LIN {X 0,Y 291.346,Z 384.19,A -85,B 0,C 180,E1 -16773.698,E2 -16773.698} C_VEL
LIN {X 0,Y 291.377,Z 384.189,A -85,B 0,C 180,E1 -16777.254,E2 -16777.254} C_VEL
LIN {X 0,Y 291.334,Z 384.196,A -85,B 0,C 180,E1 -16780.643,E2 -16780.643} C_VEL
LIN {X 0,Y 291.314,Z 384.196,A -85,B 0,C 180,E1 -16784.397,E2 -16784.397} C_VEL
LIN {X 0,Y 291.328,Z 384.196,A -85,B 0,C 180,E1 -16788.404,E2 -16788.404} C_VEL
LIN {X 0,Y 291.365,Z 384.189,A -85,B 0,C 180,E1 -16791.161,E2 -16791.161} C_VEL
LIN {X 0,Y 291.386,Z 384.191,A -85,B 0,C 180,E1 -16794.63,E2 -16794.63} C_VEL
LIN {X 0,Y 291.371,Z 384.188,A -85,B 0,C 180,E1 -16797.951,E2 -16797.951} C_VEL
LIN {X 0,Y 291.378,Z 384.187,A -85,B 0,C 180,E1 -16801.158,E2 -16801.158} C_VEL
LIN {X 0,Y 291.416,Z 384.186,A -85,B 0,C 180,E1 -16804.272,E2 -16804.272} C_VEL
LIN {X 0,Y 291.392,Z 384.185,A -85,B 0,C 180,E1 -16807.301,E2 -16807.301} C_VEL
LIN {X 0,Y 291.465,Z 384.18,A -85,B 0,C 180,E1 -16810.271,E2 -16810.271} C_VEL
LIN {X 0,Y 291.557,Z 384.166,A -85,B 0,C 180,E1 -16814.624,E2 -16814.624} C_VEL
LIN {X 0,Y 291.539,Z 384.167,A -85,B 0,C 180,E1 -16818.881,E2 -16818.881} C_VEL
LIN {X 0,Y 291.708,Z 384.147,A -85,B 0,C 180,E1 -16821.689,E2 -16821.689} C_VEL
LIN {X 0,Y 291.631,Z 384.157,A -85,B 0,C 180,E1 -16824.469,E2 -16824.469} C_VEL
LIN {X 0,Y 291.892,Z 384.124,A -85,B 0,C 180,E1 -16828.621,E2 -16828.621} C_VEL
LIN {X 0,Y 291.892,Z 384.124,A -85,B 0,C 180,E1 -16831.38,E2 -16831.38} C_VEL
LIN {X 0,Y 291.738,Z 384.142,A -85,B 0,C 180,E1 -16836.918,E2 -16836.918} C_VEL
LIN {X 0,Y 291.578,Z 384.166,A -85,B 0,C 180,E1 -16839.714,E2 -16839.714} C_VEL
LIN {X 0,Y 291.525,Z 384.172,A -85,B 0,C 180,E1 -16843.95,E2 -16843.95} C_VEL
LIN {X 0,Y 291.49,Z 384.173,A -85,B 0,C 180,E1 -16846.818,E2 -16846.818} C_VEL
LIN {X 0,Y 291.453,Z 384.18,A -85,B 0,C 180,E1 -16849.875,E2 -16849.875} C_VEL
LIN {X 0,Y 291.403,Z 384.185,A -85,B 0,C 180,E1 -16854.205,E2 -16854.205} C_VEL
LIN {X 0,Y 291.422,Z 384.184,A -85,B 0,C 180,E1 -16857.272,E2 -16857.272} C_VEL
LIN {X 0,Y 291.337,Z 384.191,A -85,B 0,C 180,E1 -16860.437,E2 -16860.437} C_VEL
LIN {X 0,Y 291.347,Z 384.194,A -85,B 0,C 180,E1 -16863.698,E2 -16863.698} C_VEL
LIN {X 0,Y 291.397,Z 384.188,A -85,B 0,C 180,E1 -16867.259,E2 -16867.259} C_VEL
LIN {X 0,Y 291.337,Z 384.192,A -85,B 0,C 180,E1 -16870.642,E2 -16870.642} C_VEL
LIN {X 0,Y 291.316,Z 384.195,A -85,B 0,C 180,E1 -16874.397,E2 -16874.397} C_VEL
LIN {X 0,Y 291.329,Z 384.193,A -85,B 0,C 180,E1 -16878.404,E2 -16878.404} C_VEL
LIN {X 0,Y 291.356,Z 384.195,A -85,B 0,C 180,E1 -16881.159,E2 -16881.159} C_VEL
LIN {X 0,Y 291.391,Z 384.186,A -85,B 0,C 180,E1 -16884.63,E2 -16884.63} C_VEL
LIN {X 0,Y 291.604,Z 384.368,A -85,B 0,C 180,E1 -16888.182,E2 -16888.182} C_VEL
LIN {X 0,Y 291.699,Z 387.226,A -85,B 0,C 180,E1 -16890.154,E2 -16890.154} C_VEL
LIN {X 0,Y 291.395,Z 391.699,A -85,B 0,C 180,E1 -16893.175,E2 -16893.175} C_VEL
LIN {X 0,Y 290.919,Z 397.87,A -85,B 0,C 180,E1 -16897.261,E2 -16897.261} C_VEL
LIN {X 0,Y 290.667,Z 402.939,A -85,B 0,C 180,E1 -16900.559,E2 -16900.559} C_VEL
LIN {X 0,Y 290.371,Z 409.272,A -85,B 0,C 180,E1 -16904.559,E2 -16904.559} C_VEL
LIN {X 0,Y 290.223,Z 413.716,A -85,B 0,C 180,E1 -16907.323,E2 -16907.323} C_VEL
LIN {X 0,Y 291.327,Z 425.543,A -85,B 0,C 180,E1 -16908.255,E2 -16908.255} C_VEL
LIN {X 0,Y 292.053,Z 433.72,A -85,B 0,C 180,E1 -16909.076,E2 -16909.076} C_VEL
LIN {X 0,Y 291.458,Z 444.808,A -85,B 0,C 180,E1 -16910.457,E2 -16910.457} C_VEL
LIN {X 0,Y 291.102,Z 453.483,A -85,B 0,C 180,E1 -16911.833,E2 -16911.833} C_VEL
LIN {X 0,Y 290.825,Z 461.477,A -85,B 0,C 180,E1 -16913.409,E2 -16913.409} C_VEL
LIN {X 0,Y 290.486,Z 468.482,A -85,B 0,C 180,E1 -16915.142,E2 -16915.142} C_VEL
LIN {X 0,Y 290.116,Z 474.952,A -85,B 0,C 180,E1 -16917.223,E2 -16917.223} C_VEL
LIN {X 0,Y 290.15,Z 479.618,A -85,B 0,C 180,E1 -16919.306,E2 -16919.306} C_VEL
LIN {X 0,Y 290.377,Z 482.726,A -85,B 0,C 180,E1 -16921.387,E2 -16921.387} C_VEL
LIN {X 0,Y 290.679,Z 483.998,A -85,B 0,C 180,E1 -16922.772,E2 -16922.772} C_VEL
LIN {X 0,Y 291.108,Z 484.656,A -85,B 0,C 180,E1 -16924.153,E2 -16924.153} C_VEL
LIN {X 0,Y 291.763,Z 484.692,A -85,B 0,C 180,E1 -16925.529,E2 -16925.529} C_VEL
LIN {X 0,Y 292.675,Z 484.009,A -85,B 0,C 180,E1 -16927.041,E2 -16927.041} C_VEL
LIN {X 0,Y 292.821,Z 483.174,A -85,B 0,C 180,E1 -16928.184,E2 -16928.184} C_VEL
LIN {X 0,Y 291.551,Z 481.327,A -85,B 0,C 180,E1 -16930.084,E2 -16930.084} C_VEL
LIN {X 0,Y 290.55,Z 478.7,A -85,B 0,C 180,E1 -16931.949,E2 -16931.949} C_VEL
LIN {X 0,Y 291.092,Z 476.418,A -85,B 0,C 180,E1 -16933.013,E2 -16933.013} C_VEL
LIN {X 0,Y 293.494,Z 470.739,A -85,B 0,C 180,E1 -16934.917,E2 -16934.917} C_VEL
LIN {X 0,Y 295.888,Z 464.445,A -85,B 0,C 180,E1 -16936.561,E2 -16936.561} C_VEL
LIN {X 0,Y 297.855,Z 458.321,A -85,B 0,C 180,E1 -16937.863,E2 -16937.863} C_VEL
LIN {X 0,Y 297.606,Z 451.062,A -85,B 0,C 180,E1 -16939.604,E2 -16939.604} C_VEL
LIN {X 0,Y 296.422,Z 443.706,A -85,B 0,C 180,E1 -16941.349,E2 -16941.349} C_VEL
LIN {X 0,Y 294.426,Z 436.045,A -85,B 0,C 180,E1 -16943.209,E2 -16943.209} C_VEL
LIN {X 0,Y 291.385,Z 427.339,A -85,B 0,C 180,E1 -16945.429,E2 -16945.429} C_VEL
LIN {X 0,Y 289.92,Z 424.703,A -85,B 0,C 180,E1 -16946.243,E2 -16946.243} C_VEL
LIN {X 0,Y 289.478,Z 422.909,A -85,B 0,C 180,E1 -16946.688,E2 -16946.688} C_VEL
LIN {X 0,Y 290.452,Z 420.929,A -85,B 0,C 180,E1 -16949.414,E2 -16949.414} C_VEL
LIN {X 0,Y 291.365,Z 419.235,A -85,B 0,C 180,E1 -16952.41,E2 -16952.41} C_VEL
LIN {X 0,Y 291.783,Z 418.234,A -85,B 0,C 180,E1 -16955.315,E2 -16955.315} C_VEL
LIN {X 0,Y 292.122,Z 417.814,A -85,B 0,C 180,E1 -16958.72,E2 -16958.72} C_VEL
LIN {X 0,Y 292.49,Z 418.223,A -85,B 0,C 180,E1 -16962.283,E2 -16962.283} C_VEL
LIN {X 0,Y 292.737,Z 418.816,A -85,B 0,C 180,E1 -16964.125,E2 -16964.125} C_VEL
LIN {X 0,Y 293.309,Z 420.913,A -85,B 0,C 180,E1 -16967.97,E2 -16967.97} C_VEL
LIN {X 0,Y 293.957,Z 423.957,A -85,B 0,C 180,E1 -16971.565,E2 -16971.565} C_VEL
LIN {X 0,Y 294.859,Z 427.941,A -85,B 0,C 180,E1 -16975.107,E2 -16975.107} C_VEL
LIN {X 0,Y 295.132,Z 430.263,A -85,B 0,C 180,E1 -16976.79,E2 -16976.79} C_VEL
LIN {X 0,Y 294.265,Z 432.986,A -85,B 0,C 180,E1 -16978.302,E2 -16978.302} C_VEL
LIN {X 0,Y 293.553,Z 434.629,A -85,B 0,C 180,E1 -16979.109,E2 -16979.109} C_VEL
LIN {X 0,Y 296.477,Z 448.571,A -85,B 0,C 180,E1 -16981.164,E2 -16981.164} C_VEL
LIN {X 0,Y 297.888,Z 460.135,A -85,B 0,C 180,E1 -16982.828,E2 -16982.828} C_VEL
LIN {X 0,Y 298.071,Z 471.015,A -85,B 0,C 180,E1 -16984.379,E2 -16984.379} C_VEL
LIN {X 0,Y 297.029,Z 480.357,A -85,B 0,C 180,E1 -16985.725,E2 -16985.725} C_VEL
LIN {X 0,Y 294.81,Z 489.886,A -85,B 0,C 180,E1 -16987.208,E2 -16987.208} C_VEL
LIN {X 0,Y 291.477,Z 500.502,A -85,B 0,C 180,E1 -16989.167,E2 -16989.167} C_VEL
LIN {X 0,Y 288.869,Z 509.05,A -85,B 0,C 180,E1 -16991.194,E2 -16991.194} C_VEL
LIN {X 0,Y 286.706,Z 516.091,A -85,B 0,C 180,E1 -16993.26,E2 -16993.26} C_VEL
LIN {X 0,Y 284.91,Z 522.618,A -85,B 0,C 180,E1 -16995.719,E2 -16995.719} C_VEL
LIN {X 0,Y 283.662,Z 527.022,A -85,B 0,C 180,E1 -16997.842,E2 -16997.842} C_VEL
LIN {X 0,Y 283.002,Z 530.416,A -85,B 0,C 180,E1 -16999.989,E2 -16999.989} C_VEL
LIN {X 0,Y 282.794,Z 532.166,A -85,B 0,C 180,E1 -17001.424,E2 -17001.424} C_VEL
LIN {X 0,Y 282.768,Z 534.128,A -85,B 0,C 180,E1 -17003.812,E2 -17003.812} C_VEL
LIN {X 0,Y 282.819,Z 534.884,A -85,B 0,C 180,E1 -17005.724,E2 -17005.724} C_VEL
LIN {X 0,Y 283.069,Z 534.95,A -85,B 0,C 180,E1 -17007.153,E2 -17007.153} C_VEL
LIN {X 0,Y 283.316,Z 534.592,A -85,B 0,C 180,E1 -17008.578,E2 -17008.578} C_VEL
LIN {X 0,Y 283.354,Z 533.788,A -85,B 0,C 180,E1 -17010,E2 -17010} C_VEL
LIN {X 0,Y 283.43,Z 532.489,A -85,B 0,C 180,E1 -17011.421,E2 -17011.421} C_VEL
LIN {X 0,Y 283.406,Z 529.608,A -85,B 0,C 180,E1 -17013.554,E2 -17013.554} C_VEL
LIN {X 0,Y 283.365,Z 525.512,A -85,B 0,C 180,E1 -17015.693,E2 -17015.693} C_VEL
LIN {X 0,Y 283.366,Z 520.078,A -85,B 0,C 180,E1 -17017.839,E2 -17017.839} C_VEL
LIN {X 0,Y 283.486,Z 513.002,A -85,B 0,C 180,E1 -17019.993,E2 -17019.993} C_VEL
LIN {X 0,Y 283.859,Z 505.706,A -85,B 0,C 180,E1 -17021.786,E2 -17021.786} C_VEL
LIN {X 0,Y 284.405,Z 496.736,A -85,B 0,C 180,E1 -17023.577,E2 -17023.577} C_VEL
LIN {X 0,Y 285.267,Z 485.479,A -85,B 0,C 180,E1 -17025.357,E2 -17025.357} C_VEL
LIN {X 0,Y 286.009,Z 474.805,A -85,B 0,C 180,E1 -17026.679,E2 -17026.679} C_VEL
LIN {X 0,Y 285.534,Z 465.102,A -85,B 0,C 180,E1 -17027.641,E2 -17027.641} C_VEL
LIN {X 0,Y 284.705,Z 452.326,A -85,B 0,C 180,E1 -17028.624,E2 -17028.624} C_VEL
LIN {X 0,Y 284.322,Z 438.684,A -85,B 0,C 180,E1 -17029.352,E2 -17029.352} C_VEL
LIN {X 0,Y 286.278,Z 425.026,A -85,B 0,C 180,E1 -17034.723,E2 -17034.723} C_VEL
LIN {X 0,Y 288.392,Z 413.702,A -85,B 0,C 180,E1 -17039.169,E2 -17039.169} C_VEL
LIN {X 0,Y 289.2,Z 409.854,A -85,B 0,C 180,E1 -17040.686,E2 -17040.686} C_VEL
LIN {X 0,Y 288.584,Z 405.721,A -85,B 0,C 180,E1 -17042.396,E2 -17042.396} C_VEL
LIN {X 0,Y 286.392,Z 395.189,A -85,B 0,C 180,E1 -17046.957,E2 -17046.957} C_VEL
LIN {X 0,Y 284.562,Z 386.236,A -85,B 0,C 180,E1 -17051.05,E2 -17051.05} C_VEL
LIN {X 0,Y 284.311,Z 385.071,A -85,B 0,C 180,E1 -17051.685,E2 -17051.685} C_VEL
LIN {X 0,Y 284.266,Z 385.073,A -85,B 0,C 180,E1 -17055.805,E2 -17055.805} C_VEL
LIN {X 0,Y 284.307,Z 385.071,A -85,B 0,C 180,E1 -17060.024,E2 -17060.024} C_VEL
LIN {X 0,Y 284.351,Z 385.064,A -85,B 0,C 180,E1 -17063.617,E2 -17063.617} C_VEL
LIN {X 0,Y 284.308,Z 385.067,A -85,B 0,C 180,E1 -17067.189,E2 -17067.189} C_VEL
LIN {X 0,Y 284.356,Z 385.064,A -85,B 0,C 180,E1 -17070.376,E2 -17070.376} C_VEL
LIN {X 0,Y 284.378,Z 385.06,A -85,B 0,C 180,E1 -17073.587,E2 -17073.587} C_VEL
LIN {X 0,Y 284.367,Z 385.06,A -85,B 0,C 180,E1 -17076.707,E2 -17076.707} C_VEL
LIN {X 0,Y 284.404,Z 385.056,A -85,B 0,C 180,E1 -17081.262,E2 -17081.262} C_VEL
LIN {X 0,Y 284.493,Z 385.045,A -85,B 0,C 180,E1 -17084.459,E2 -17084.459} C_VEL
LIN {X 0,Y 284.489,Z 385.045,A -85,B 0,C 180,E1 -17088.601,E2 -17088.601} C_VEL
LIN {X 0,Y 284.66,Z 385.026,A -85,B 0,C 180,E1 -17091.481,E2 -17091.481} C_VEL
LIN {X 0,Y 284.603,Z 385.031,A -85,B 0,C 180,E1 -17094.331,E2 -17094.331} C_VEL
LIN {X 0,Y 284.859,Z 384.998,A -85,B 0,C 180,E1 -17098.586,E2 -17098.586} C_VEL
LIN {X 0,Y 284.856,Z 385.003,A -85,B 0,C 180,E1 -17101.414,E2 -17101.414} C_VEL
LIN {X 0,Y 284.699,Z 385.021,A -85,B 0,C 180,E1 -17107.09,E2 -17107.09} C_VEL
LIN {X 0,Y 284.568,Z 385.036,A -85,B 0,C 180,E1 -17109.955,E2 -17109.955} C_VEL
LIN {X 0,Y 284.483,Z 385.046,A -85,B 0,C 180,E1 -17114.303,E2 -17114.303} C_VEL
LIN {X 0,Y 284.426,Z 385.057,A -85,B 0,C 180,E1 -17117.248,E2 -17117.248} C_VEL
LIN {X 0,Y 284.379,Z 385.059,A -85,B 0,C 180,E1 -17120.242,E2 -17120.242} C_VEL
LIN {X 0,Y 284.37,Z 385.06,A -85,B 0,C 180,E1 -17123.876,E2 -17123.876} C_VEL
LIN {X 0,Y 284.398,Z 385.06,A -85,B 0,C 180,E1 -17127.174,E2 -17127.174} C_VEL
LIN {X 0,Y 284.297,Z 385.071,A -85,B 0,C 180,E1 -17131.274,E2 -17131.274} C_VEL
LIN {X 0,Y 284.341,Z 385.065,A -85,B 0,C 180,E1 -17135.348,E2 -17135.348} C_VEL
LIN {X 0,Y 284.313,Z 385.068,A -85,B 0,C 180,E1 -17138.169,E2 -17138.169} C_VEL
LIN {X 0,Y 284.27,Z 385.072,A -85,B 0,C 180,E1 -17142.125,E2 -17142.125} C_VEL
LIN {X 0,Y 284.269,Z 385.073,A -85,B 0,C 180,E1 -17146.192,E2 -17146.192} C_VEL
LIN {X 0,Y 284.308,Z 385.068,A -85,B 0,C 180,E1 -17150.024,E2 -17150.024} C_VEL
LIN {X 0,Y 284.351,Z 385.062,A -85,B 0,C 180,E1 -17153.617,E2 -17153.617} C_VEL
LIN {X 0,Y 284.308,Z 385.068,A -85,B 0,C 180,E1 -17157.19,E2 -17157.19} C_VEL
LIN {X 0,Y 284.356,Z 385.065,A -85,B 0,C 180,E1 -17160.376,E2 -17160.376} C_VEL
LIN {X 0,Y 284.377,Z 385.059,A -85,B 0,C 180,E1 -17163.587,E2 -17163.587} C_VEL
LIN {X 0,Y 284.371,Z 385.061,A -85,B 0,C 180,E1 -17166.708,E2 -17166.708} C_VEL
LIN {X 0,Y 284.408,Z 385.055,A -85,B 0,C 180,E1 -17171.262,E2 -17171.262} C_VEL
LIN {X 0,Y 284.495,Z 385.047,A -85,B 0,C 180,E1 -17174.459,E2 -17174.459} C_VEL
LIN {X 0,Y 284.491,Z 385.046,A -85,B 0,C 180,E1 -17178.602,E2 -17178.602} C_VEL
LIN {X 0,Y 284.659,Z 385.025,A -85,B 0,C 180,E1 -17181.481,E2 -17181.481} C_VEL
LIN {X 0,Y 284.601,Z 385.033,A -85,B 0,C 180,E1 -17184.332,E2 -17184.332} C_VEL
LIN {X 0,Y 284.858,Z 385,A -85,B 0,C 180,E1 -17188.587,E2 -17188.587} C_VEL
LIN {X 0,Y 284.858,Z 385,A -85,B 0,C 180,E1 -17191.414,E2 -17191.414} C_VEL
LIN {X 0,Y 284.689,Z 385.02,A -85,B 0,C 180,E1 -17197.091,E2 -17197.091} C_VEL
LIN {X 0,Y 284.522,Z 385.045,A -85,B 0,C 180,E1 -17199.957,E2 -17199.957} C_VEL
LIN {X 0,Y 284.484,Z 385.046,A -85,B 0,C 180,E1 -17204.303,E2 -17204.303} C_VEL
LIN {X 0,Y 284.428,Z 385.054,A -85,B 0,C 180,E1 -17207.248,E2 -17207.248} C_VEL
LIN {X 0,Y 284.383,Z 385.058,A -85,B 0,C 180,E1 -17210.242,E2 -17210.242} C_VEL
LIN {X 0,Y 284.372,Z 385.062,A -85,B 0,C 180,E1 -17213.876,E2 -17213.876} C_VEL
LIN {X 0,Y 284.398,Z 385.059,A -85,B 0,C 180,E1 -17217.173,E2 -17217.173} C_VEL
LIN {X 0,Y 284.296,Z 385.071,A -85,B 0,C 180,E1 -17221.275,E2 -17221.275} C_VEL
LIN {X 0,Y 284.364,Z 385.065,A -85,B 0,C 180,E1 -17225.354,E2 -17225.354} C_VEL
LIN {X 0,Y 284.326,Z 385.064,A -85,B 0,C 180,E1 -17228.167,E2 -17228.167} C_VEL
LIN {X 0,Y 284.272,Z 385.072,A -85,B 0,C 180,E1 -17232.125,E2 -17232.125} C_VEL
LIN {X 0,Y 284.271,Z 385.071,A -85,B 0,C 180,E1 -17236.192,E2 -17236.192} C_VEL
LIN {X 0,Y 284.309,Z 385.068,A -85,B 0,C 180,E1 -17240.024,E2 -17240.024} C_VEL
LIN {X 0,Y 284.345,Z 385.064,A -85,B 0,C 180,E1 -17243.616,E2 -17243.616} C_VEL
LIN {X 0,Y 284.551,Z 385.237,A -85,B 0,C 180,E1 -17248.134,E2 -17248.134} C_VEL
LIN {X 0,Y 284.632,Z 388.458,A -85,B 0,C 180,E1 -17250.407,E2 -17250.407} C_VEL
LIN {X 0,Y 284.263,Z 393.091,A -85,B 0,C 180,E1 -17253.575,E2 -17253.575} C_VEL
LIN {X 0,Y 283.836,Z 398.85,A -85,B 0,C 180,E1 -17257.431,E2 -17257.431} C_VEL
LIN {X 0,Y 283.535,Z 404.576,A -85,B 0,C 180,E1 -17261.202,E2 -17261.202} C_VEL
LIN {X 0,Y 283.229,Z 411.459,A -85,B 0,C 180,E1 -17265.633,E2 -17265.633} C_VEL
LIN {X 0,Y 283.144,Z 414.142,A -85,B 0,C 180,E1 -17267.274,E2 -17267.274} C_VEL
LIN {X 0,Y 284.263,Z 426.11,A -85,B 0,C 180,E1 -17268.231,E2 -17268.231} C_VEL
LIN {X 0,Y 284.981,Z 433.465,A -85,B 0,C 180,E1 -17268.981,E2 -17268.981} C_VEL
LIN {X 0,Y 284.481,Z 443.471,A -85,B 0,C 180,E1 -17270.221,E2 -17270.221} C_VEL
LIN {X 0,Y 284.044,Z 453.067,A -85,B 0,C 180,E1 -17271.724,E2 -17271.724} C_VEL
LIN {X 0,Y 283.74,Z 460.853,A -85,B 0,C 180,E1 -17273.243,E2 -17273.243} C_VEL
LIN {X 0,Y 283.422,Z 468.151,A -85,B 0,C 180,E1 -17275.021,E2 -17275.021} C_VEL
LIN {X 0,Y 283.079,Z 473.868,A -85,B 0,C 180,E1 -17276.798,E2 -17276.798} C_VEL
LIN {X 0,Y 283.01,Z 478.297,A -85,B 0,C 180,E1 -17278.577,E2 -17278.577} C_VEL
LIN {X 0,Y 283.2,Z 482.167,A -85,B 0,C 180,E1 -17280.711,E2 -17280.711} C_VEL
LIN {X 0,Y 283.618,Z 484.578,A -85,B 0,C 180,E1 -17282.841,E2 -17282.841} C_VEL
LIN {X 0,Y 284.09,Z 485.407,A -85,B 0,C 180,E1 -17284.256,E2 -17284.256} C_VEL
LIN {X 0,Y 284.756,Z 485.606,A -85,B 0,C 180,E1 -17285.666,E2 -17285.666} C_VEL
LIN {X 0,Y 285.739,Z 485.062,A -85,B 0,C 180,E1 -17287.255,E2 -17287.255} C_VEL
LIN {X 0,Y 286.62,Z 484.196,A -85,B 0,C 180,E1 -17288.46,E2 -17288.46} C_VEL
LIN {X 0,Y 288.505,Z 481.559,A -85,B 0,C 180,E1 -17290.527,E2 -17290.527} C_VEL
LIN {X 0,Y 290.577,Z 477.527,A -85,B 0,C 180,E1 -17292.573,E2 -17292.573} C_VEL
LIN {X 0,Y 291.092,Z 476.418,A -85,B 0,C 180,E1 -17293.013,E2 -17293.013} C_VEL
LIN {X 0,Y 291.836,Z 473.847,A -85,B 0,C 180,E1 -17294.043,E2 -17294.043} C_VEL
LIN {X 0,Y 291.733,Z 469.418,A -85,B 0,C 180,E1 -17295.769,E2 -17295.769} C_VEL
LIN {X 0,Y 291.411,Z 463.289,A -85,B 0,C 180,E1 -17297.763,E2 -17297.763} C_VEL
LIN {X 0,Y 291.7,Z 460.914,A -85,B 0,C 180,E1 -17298.38,E2 -17298.38} C_VEL
LIN {X 0,Y 291.886,Z 455.82,A -85,B 0,C 180,E1 -17299.7,E2 -17299.7} C_VEL
LIN {X 0,Y 290.962,Z 447.353,A -85,B 0,C 180,E1 -17301.873,E2 -17301.873} C_VEL
LIN {X 0,Y 289.143,Z 439.574,A -85,B 0,C 180,E1 -17303.919,E2 -17303.919} C_VEL
LIN {X 0,Y 286.986,Z 432.608,A -85,B 0,C 180,E1 -17305.847,E2 -17305.847} C_VEL
LIN {X 0,Y 284.956,Z 427.727,A -85,B 0,C 180,E1 -17307.391,E2 -17307.391} C_VEL
LIN {X 0,Y 283.978,Z 425.851,A -85,B 0,C 180,E1 -17308.049,E2 -17308.049} C_VEL
LIN {X 0,Y 283.409,Z 423.808,A -85,B 0,C 180,E1 -17308.615,E2 -17308.615} C_VEL
LIN {X 0,Y 284.296,Z 422.222,A -85,B 0,C 180,E1 -17311.274,E2 -17311.274} C_VEL
LIN {X 0,Y 284.754,Z 421.435,A -85,B 0,C 180,E1 -17312.948,E2 -17312.948} C_VEL
LIN {X 0,Y 285.231,Z 420.555,A -85,B 0,C 180,E1 -17316.253,E2 -17316.253} C_VEL
LIN {X 0,Y 285.619,Z 420.397,A -85,B 0,C 180,E1 -17319.774,E2 -17319.774} C_VEL
LIN {X 0,Y 286.041,Z 421.202,A -85,B 0,C 180,E1 -17323.469,E2 -17323.469} C_VEL
LIN {X 0,Y 286.58,Z 423.127,A -85,B 0,C 180,E1 -17327.368,E2 -17327.368} C_VEL
LIN {X 0,Y 287.095,Z 425.487,A -85,B 0,C 180,E1 -17330.47,E2 -17330.47} C_VEL
LIN {X 0,Y 287.965,Z 429.258,A -85,B 0,C 180,E1 -17334.144,E2 -17334.144} C_VEL
LIN {X 0,Y 288.365,Z 432.715,A -85,B 0,C 180,E1 -17336.777,E2 -17336.777} C_VEL
LIN {X 0,Y 288.004,Z 434.072,A -85,B 0,C 180,E1 -17337.53,E2 -17337.53} C_VEL
LIN {X 0,Y 290.818,Z 447.57,A -85,B 0,C 180,E1 -17339.771,E2 -17339.771} C_VEL
LIN {X 0,Y 292.302,Z 461.035,A -85,B 0,C 180,E1 -17341.869,E2 -17341.869} C_VEL
LIN {X 0,Y 292.319,Z 470.96,A -85,B 0,C 180,E1 -17343.388,E2 -17343.388} C_VEL
LIN {X 0,Y 291.244,Z 480.275,A -85,B 0,C 180,E1 -17344.829,E2 -17344.829} C_VEL
LIN {X 0,Y 289.005,Z 489.552,A -85,B 0,C 180,E1 -17346.344,E2 -17346.344} C_VEL
LIN {X 0,Y 286.069,Z 498.391,A -85,B 0,C 180,E1 -17347.997,E2 -17347.997} C_VEL
LIN {X 0,Y 283.584,Z 505.824,A -85,B 0,C 180,E1 -17349.698,E2 -17349.698} C_VEL
LIN {X 0,Y 280.909,Z 513.434,A -85,B 0,C 180,E1 -17351.851,E2 -17351.851} C_VEL
LIN {X 0,Y 278.979,Z 519.262,A -85,B 0,C 180,E1 -17353.912,E2 -17353.912} C_VEL
LIN {X 0,Y 277.52,Z 524.166,A -85,B 0,C 180,E1 -17356.079,E2 -17356.079} C_VEL
LIN {X 0,Y 276.348,Z 528.017,A -85,B 0,C 180,E1 -17358.261,E2 -17358.261} C_VEL
LIN {X 0,Y 275.948,Z 530.063,A -85,B 0,C 180,E1 -17359.73,E2 -17359.73} C_VEL
LIN {X 0,Y 275.681,Z 532.878,A -85,B 0,C 180,E1 -17362.676,E2 -17362.676} C_VEL
LIN {X 0,Y 275.707,Z 533.703,A -85,B 0,C 180,E1 -17364.147,E2 -17364.147} C_VEL
LIN {X 0,Y 276.004,Z 534.05,A -85,B 0,C 180,E1 -17367.081,E2 -17367.081} C_VEL
LIN {X 0,Y 276.27,Z 533.623,A -85,B 0,C 180,E1 -17368.542,E2 -17368.542} C_VEL
LIN {X 0,Y 276.338,Z 532.687,A -85,B 0,C 180,E1 -17370,E2 -17370} C_VEL
LIN {X 0,Y 276.415,Z 531.297,A -85,B 0,C 180,E1 -17371.457,E2 -17371.457} C_VEL
LIN {X 0,Y 276.406,Z 528.256,A -85,B 0,C 180,E1 -17373.644,E2 -17373.644} C_VEL
LIN {X 0,Y 276.363,Z 523.98,A -85,B 0,C 180,E1 -17375.838,E2 -17375.838} C_VEL
LIN {X 0,Y 276.344,Z 518.268,A -85,B 0,C 180,E1 -17378.04,E2 -17378.04} C_VEL
LIN {X 0,Y 276.513,Z 510.973,A -85,B 0,C 180,E1 -17380.248,E2 -17380.248} C_VEL
LIN {X 0,Y 276.88,Z 503.352,A -85,B 0,C 180,E1 -17382.087,E2 -17382.087} C_VEL
LIN {X 0,Y 277.417,Z 494.985,A -85,B 0,C 180,E1 -17383.739,E2 -17383.739} C_VEL
LIN {X 0,Y 278.218,Z 484.775,A -85,B 0,C 180,E1 -17385.381,E2 -17385.381} C_VEL
LIN {X 0,Y 278.942,Z 473.704,A -85,B 0,C 180,E1 -17386.78,E2 -17386.78} C_VEL
LIN {X 0,Y 278.239,Z 462.1,A -85,B 0,C 180,E1 -17387.929,E2 -17387.929} C_VEL
LIN {X 0,Y 277.496,Z 449.034,A -85,B 0,C 180,E1 -17388.887,E2 -17388.887} C_VEL
LIN {X 0,Y 277.262,Z 438.473,A -85,B 0,C 180,E1 -17389.448,E2 -17389.448} C_VEL
LIN {X 0,Y 279.313,Z 424.599,A -85,B 0,C 180,E1 -17395.065,E2 -17395.065} C_VEL
LIN {X 0,Y 281.704,Z 412.566,A -85,B 0,C 180,E1 -17399.931,E2 -17399.931} C_VEL
LIN {X 0,Y 282.109,Z 409.634,A -85,B 0,C 180,E1 -17401.126,E2 -17401.126} C_VEL
LIN {X 0,Y 280.171,Z 400.291,A -85,B 0,C 180,E1 -17405.236,E2 -17405.236} C_VEL
LIN {X 0,Y 278.436,Z 391.787,A -85,B 0,C 180,E1 -17409.125,E2 -17409.125} C_VEL
LIN {X 0,Y 277.278,Z 385.948,A -85,B 0,C 180,E1 -17411.974,E2 -17411.974} C_VEL
LIN {X 0,Y 277.22,Z 385.949,A -85,B 0,C 180,E1 -17415.222,E2 -17415.222} C_VEL
LIN {X 0,Y 277.223,Z 385.95,A -85,B 0,C 180,E1 -17419.512,E2 -17419.512} C_VEL
LIN {X 0,Y 277.282,Z 385.945,A -85,B 0,C 180,E1 -17422.533,E2 -17422.533} C_VEL
LIN {X 0,Y 277.254,Z 385.95,A -85,B 0,C 180,E1 -17426.105,E2 -17426.105} C_VEL
LIN {X 0,Y 277.262,Z 385.947,A -85,B 0,C 180,E1 -17429.538,E2 -17429.538} C_VEL
LIN {X 0,Y 277.358,Z 385.933,A -85,B 0,C 180,E1 -17432.864,E2 -17432.864} C_VEL
LIN {X 0,Y 277.329,Z 385.94,A -85,B 0,C 180,E1 -17436.08,E2 -17436.08} C_VEL
LIN {X 0,Y 277.346,Z 385.935,A -85,B 0,C 180,E1 -17440.766,E2 -17440.766} C_VEL
LIN {X 0,Y 277.435,Z 385.925,A -85,B 0,C 180,E1 -17445.326,E2 -17445.326} C_VEL
LIN {X 0,Y 277.507,Z 385.918,A -85,B 0,C 180,E1 -17449.789,E2 -17449.789} C_VEL
LIN {X 0,Y 277.654,Z 385.896,A -85,B 0,C 180,E1 -17452.729,E2 -17452.729} C_VEL
LIN {X 0,Y 277.825,Z 385.875,A -85,B 0,C 180,E1 -17458.55,E2 -17458.55} C_VEL
LIN {X 0,Y 277.822,Z 385.879,A -85,B 0,C 180,E1 -17461.45,E2 -17461.45} C_VEL
LIN {X 0,Y 277.654,Z 385.9,A -85,B 0,C 180,E1 -17467.271,E2 -17467.271} C_VEL
LIN {X 0,Y 277.508,Z 385.914,A -85,B 0,C 180,E1 -17470.211,E2 -17470.211} C_VEL
LIN {X 0,Y 277.436,Z 385.924,A -85,B 0,C 180,E1 -17474.674,E2 -17474.674} C_VEL
LIN {X 0,Y 277.346,Z 385.939,A -85,B 0,C 180,E1 -17479.234,E2 -17479.234} C_VEL
LIN {X 0,Y 277.32,Z 385.938,A -85,B 0,C 180,E1 -17484.171,E2 -17484.171} C_VEL
LIN {X 0,Y 277.326,Z 385.939,A -85,B 0,C 180,E1 -17487.505,E2 -17487.505} C_VEL
LIN {X 0,Y 277.272,Z 385.945,A -85,B 0,C 180,E1 -17490.482,E2 -17490.482} C_VEL
LIN {X 0,Y 277.247,Z 385.946,A -85,B 0,C 180,E1 -17493.896,E2 -17493.896} C_VEL
LIN {X 0,Y 277.268,Z 385.945,A -85,B 0,C 180,E1 -17497.469,E2 -17497.469} C_VEL
LIN {X 0,Y 277.21,Z 385.953,A -85,B 0,C 180,E1 -17501.237,E2 -17501.237} C_VEL
LIN {X 0,Y 277.217,Z 385.952,A -85,B 0,C 180,E1 -17505.223,E2 -17505.223} C_VEL
LIN {X 0,Y 277.223,Z 385.95,A -85,B 0,C 180,E1 -17509.512,E2 -17509.512} C_VEL
LIN {X 0,Y 277.283,Z 385.945,A -85,B 0,C 180,E1 -17512.533,E2 -17512.533} C_VEL
LIN {X 0,Y 277.255,Z 385.948,A -85,B 0,C 180,E1 -17516.106,E2 -17516.106} C_VEL
LIN {X 0,Y 277.262,Z 385.944,A -85,B 0,C 180,E1 -17519.539,E2 -17519.539} C_VEL
LIN {X 0,Y 277.358,Z 385.935,A -85,B 0,C 180,E1 -17522.864,E2 -17522.864} C_VEL
LIN {X 0,Y 277.331,Z 385.939,A -85,B 0,C 180,E1 -17526.08,E2 -17526.08} C_VEL
LIN {X 0,Y 277.349,Z 385.936,A -85,B 0,C 180,E1 -17530.767,E2 -17530.767} C_VEL
LIN {X 0,Y 277.439,Z 385.923,A -85,B 0,C 180,E1 -17535.326,E2 -17535.326} C_VEL
LIN {X 0,Y 277.509,Z 385.916,A -85,B 0,C 180,E1 -17539.789,E2 -17539.789} C_VEL
LIN {X 0,Y 277.652,Z 385.897,A -85,B 0,C 180,E1 -17542.729,E2 -17542.729} C_VEL
LIN {X 0,Y 277.824,Z 385.876,A -85,B 0,C 180,E1 -17548.551,E2 -17548.551} C_VEL
LIN {X 0,Y 277.824,Z 385.876,A -85,B 0,C 180,E1 -17551.45,E2 -17551.45} C_VEL
LIN {X 0,Y 277.644,Z 385.898,A -85,B 0,C 180,E1 -17557.271,E2 -17557.271} C_VEL
LIN {X 0,Y 277.464,Z 385.922,A -85,B 0,C 180,E1 -17560.213,E2 -17560.213} C_VEL
LIN {X 0,Y 277.437,Z 385.923,A -85,B 0,C 180,E1 -17564.674,E2 -17564.674} C_VEL
LIN {X 0,Y 277.348,Z 385.936,A -85,B 0,C 180,E1 -17569.234,E2 -17569.234} C_VEL
LIN {X 0,Y 277.332,Z 385.939,A -85,B 0,C 180,E1 -17573.921,E2 -17573.921} C_VEL
LIN {X 0,Y 277.326,Z 385.942,A -85,B 0,C 180,E1 -17577.505,E2 -17577.505} C_VEL
LIN {X 0,Y 277.274,Z 385.943,A -85,B 0,C 180,E1 -17580.482,E2 -17580.482} C_VEL
LIN {X 0,Y 277.256,Z 385.948,A -85,B 0,C 180,E1 -17583.895,E2 -17583.895} C_VEL
LIN {X 0,Y 277.284,Z 385.945,A -85,B 0,C 180,E1 -17587.467,E2 -17587.467} C_VEL
LIN {X 0,Y 277.212,Z 385.955,A -85,B 0,C 180,E1 -17591.237,E2 -17591.237} C_VEL
LIN {X 0,Y 277.219,Z 385.955,A -85,B 0,C 180,E1 -17595.223,E2 -17595.223} C_VEL
LIN {X 0,Y 277.225,Z 385.952,A -85,B 0,C 180,E1 -17599.512,E2 -17599.512} C_VEL
LIN {X 0,Y 277.273,Z 385.945,A -85,B 0,C 180,E1 -17602.531,E2 -17602.531} C_VEL
LIN {X 0,Y 277.35,Z 385.935,A -85,B 0,C 180,E1 -17606.743,E2 -17606.743} C_VEL
LIN {X 0,Y 277.491,Z 386.108,A -85,B 0,C 180,E1 -17608.074,E2 -17608.074} C_VEL
LIN {X 0,Y 277.662,Z 388.205,A -85,B 0,C 180,E1 -17609.587,E2 -17609.587} C_VEL
LIN {X 0,Y 277.326,Z 392.869,A -85,B 0,C 180,E1 -17612.861,E2 -17612.861} C_VEL
LIN {X 0,Y 276.82,Z 398.646,A -85,B 0,C 180,E1 -17616.826,E2 -17616.826} C_VEL
LIN {X 0,Y 276.498,Z 404.429,A -85,B 0,C 180,E1 -17620.705,E2 -17620.705} C_VEL
LIN {X 0,Y 276.202,Z 410.21,A -85,B 0,C 180,E1 -17624.504,E2 -17624.504} C_VEL
LIN {X 0,Y 276.063,Z 414.35,A -85,B 0,C 180,E1 -17627.176,E2 -17627.176} C_VEL
LIN {X 0,Y 277.192,Z 426.674,A -85,B 0,C 180,E1 -17628.204,E2 -17628.204} C_VEL
LIN {X 0,Y 277.878,Z 433.193,A -85,B 0,C 180,E1 -17628.881,E2 -17628.881} C_VEL
LIN {X 0,Y 277.403,Z 443.381,A -85,B 0,C 180,E1 -17630.153,E2 -17630.153} C_VEL
LIN {X 0,Y 276.997,Z 452.264,A -85,B 0,C 180,E1 -17631.543,E2 -17631.543} C_VEL
LIN {X 0,Y 276.659,Z 460.106,A -85,B 0,C 180,E1 -17633.069,E2 -17633.069} C_VEL
LIN {X 0,Y 276.364,Z 467.661,A -85,B 0,C 180,E1 -17634.894,E2 -17634.894} C_VEL
LIN {X 0,Y 275.946,Z 474.682,A -85,B 0,C 180,E1 -17637.08,E2 -17637.08} C_VEL
LIN {X 0,Y 275.978,Z 479.889,A -85,B 0,C 180,E1 -17639.27,E2 -17639.27} C_VEL
LIN {X 0,Y 276.248,Z 483.495,A -85,B 0,C 180,E1 -17641.458,E2 -17641.458} C_VEL
LIN {X 0,Y 276.56,Z 485.092,A -85,B 0,C 180,E1 -17642.913,E2 -17642.913} C_VEL
LIN {X 0,Y 277.055,Z 486.079,A -85,B 0,C 180,E1 -17644.364,E2 -17644.364} C_VEL
LIN {X 0,Y 277.751,Z 486.463,A -85,B 0,C 180,E1 -17645.809,E2 -17645.809} C_VEL
LIN {X 0,Y 278.646,Z 486.248,A -85,B 0,C 180,E1 -17647.245,E2 -17647.245} C_VEL
LIN {X 0,Y 279.705,Z 485.441,A -85,B 0,C 180,E1 -17648.671,E2 -17648.671} C_VEL
LIN {X 0,Y 281.696,Z 483.079,A -85,B 0,C 180,E1 -17650.785,E2 -17650.785} C_VEL
LIN {X 0,Y 283.857,Z 479.349,A -85,B 0,C 180,E1 -17652.875,E2 -17652.875} C_VEL
LIN {X 0,Y 286.45,Z 474.156,A -85,B 0,C 180,E1 -17654.929,E2 -17654.929} C_VEL
LIN {X 0,Y 288.909,Z 468.504,A -85,B 0,C 180,E1 -17656.609,E2 -17656.609} C_VEL
LIN {X 0,Y 291.7,Z 460.914,A -85,B 0,C 180,E1 -17658.38,E2 -17658.38} C_VEL
LIN {X 0,Y 291.768,Z 458.619,A -85,B 0,C 180,E1 -17659.001,E2 -17659.001} C_VEL
LIN {X 0,Y 290.776,Z 455.722,A -85,B 0,C 180,E1 -17659.995,E2 -17659.995} C_VEL
LIN {X 0,Y 285.318,Z 448.239,A -85,B 0,C 180,E1 -17663.107,E2 -17663.107} C_VEL
LIN {X 0,Y 284.629,Z 446.126,A -85,B 0,C 180,E1 -17663.788,E2 -17663.788} C_VEL
LIN {X 0,Y 282.424,Z 437.433,A -85,B 0,C 180,E1 -17666.382,E2 -17666.382} C_VEL
LIN {X 0,Y 281.253,Z 433.862,A -85,B 0,C 180,E1 -17667.535,E2 -17667.535} C_VEL
LIN {X 0,Y 279.359,Z 429.098,A -85,B 0,C 180,E1 -17669.271,E2 -17669.271} C_VEL
LIN {X 0,Y 277.751,Z 425.837,A -85,B 0,C 180,E1 -17670.648,E2 -17670.648} C_VEL
LIN {X 0,Y 277.515,Z 424.772,A -85,B 0,C 180,E1 -17671.05,E2 -17671.05} C_VEL
LIN {X 0,Y 278.208,Z 423.653,A -85,B 0,C 180,E1 -17673.763,E2 -17673.763} C_VEL
LIN {X 0,Y 278.585,Z 423.1,A -85,B 0,C 180,E1 -17676.168,E2 -17676.168} C_VEL
LIN {X 0,Y 278.891,Z 422.96,A -85,B 0,C 180,E1 -17679.05,E2 -17679.05} C_VEL
LIN {X 0,Y 279.368,Z 423.592,A -85,B 0,C 180,E1 -17682.784,E2 -17682.784} C_VEL
LIN {X 0,Y 279.882,Z 425.349,A -85,B 0,C 180,E1 -17686.736,E2 -17686.736} C_VEL
LIN {X 0,Y 280.312,Z 427.122,A -85,B 0,C 180,E1 -17689.316,E2 -17689.316} C_VEL
LIN {X 0,Y 281.058,Z 430.656,A -85,B 0,C 180,E1 -17693.147,E2 -17693.147} C_VEL
LIN {X 0,Y 281.642,Z 433.418,A -85,B 0,C 180,E1 -17695.383,E2 -17695.383} C_VEL
LIN {X 0,Y 283.578,Z 438.057,A -85,B 0,C 180,E1 -17696.626,E2 -17696.626} C_VEL
LIN {X 0,Y 285.414,Z 447.46,A -85,B 0,C 180,E1 -17698.384,E2 -17698.384} C_VEL
LIN {X 0,Y 286.667,Z 459.662,A -85,B 0,C 180,E1 -17700.465,E2 -17700.465} C_VEL
LIN {X 0,Y 286.74,Z 470.393,A -85,B 0,C 180,E1 -17702.245,E2 -17702.245} C_VEL
LIN {X 0,Y 285.742,Z 479.369,A -85,B 0,C 180,E1 -17703.722,E2 -17703.722} C_VEL
LIN {X 0,Y 283.247,Z 489.377,A -85,B 0,C 180,E1 -17705.442,E2 -17705.442} C_VEL
LIN {X 0,Y 280.192,Z 498.046,A -85,B 0,C 180,E1 -17707.121,E2 -17707.121} C_VEL
LIN {X 0,Y 277.99,Z 503.959,A -85,B 0,C 180,E1 -17708.495,E2 -17708.495} C_VEL
LIN {X 0,Y 275.108,Z 511.518,A -85,B 0,C 180,E1 -17710.603,E2 -17710.603} C_VEL
LIN {X 0,Y 272.802,Z 517.677,A -85,B 0,C 180,E1 -17712.766,E2 -17712.766} C_VEL
LIN {X 0,Y 271.127,Z 522.685,A -85,B 0,C 180,E1 -17714.976,E2 -17714.976} C_VEL
LIN {X 0,Y 269.72,Z 526.65,A -85,B 0,C 180,E1 -17717.204,E2 -17717.204} C_VEL
LIN {X 0,Y 268.914,Z 529.655,A -85,B 0,C 180,E1 -17719.458,E2 -17719.458} C_VEL
LIN {X 0,Y 268.606,Z 532.276,A -85,B 0,C 180,E1 -17722.483,E2 -17722.483} C_VEL
LIN {X 0,Y 268.649,Z 532.958,A -85,B 0,C 180,E1 -17723.993,E2 -17723.993} C_VEL
LIN {X 0,Y 268.941,Z 533.136,A -85,B 0,C 180,E1 -17727.004,E2 -17727.004} C_VEL
LIN {X 0,Y 269.236,Z 532.573,A -85,B 0,C 180,E1 -17728.504,E2 -17728.504} C_VEL
LIN {X 0,Y 269.326,Z 531.549,A -85,B 0,C 180,E1 -17730,E2 -17730} C_VEL
LIN {X 0,Y 269.405,Z 529.107,A -85,B 0,C 180,E1 -17732.242,E2 -17732.242} C_VEL
LIN {X 0,Y 269.378,Z 525.487,A -85,B 0,C 180,E1 -17734.489,E2 -17734.489} C_VEL
LIN {X 0,Y 269.353,Z 520.132,A -85,B 0,C 180,E1 -17736.896,E2 -17736.896} C_VEL
LIN {X 0,Y 269.382,Z 514.048,A -85,B 0,C 180,E1 -17739.006,E2 -17739.006} C_VEL
LIN {X 0,Y 269.632,Z 507.318,A -85,B 0,C 180,E1 -17740.893,E2 -17740.893} C_VEL
LIN {X 0,Y 270.111,Z 499.06,A -85,B 0,C 180,E1 -17742.777,E2 -17742.777} C_VEL
LIN {X 0,Y 270.757,Z 488.774,A -85,B 0,C 180,E1 -17744.66,E2 -17744.66} C_VEL
LIN {X 0,Y 271.551,Z 478.517,A -85,B 0,C 180,E1 -17746.154,E2 -17746.154} C_VEL
LIN {X 0,Y 271.803,Z 472.185,A -85,B 0,C 180,E1 -17746.92,E2 -17746.92} C_VEL
LIN {X 0,Y 270.97,Z 459.849,A -85,B 0,C 180,E1 -17748.134,E2 -17748.134} C_VEL
LIN {X 0,Y 270.301,Z 447.101,A -85,B 0,C 180,E1 -17749.064,E2 -17749.064} C_VEL
LIN {X 0,Y 270.199,Z 438.12,A -85,B 0,C 180,E1 -17749.565,E2 -17749.565} C_VEL
LIN {X 0,Y 272.322,Z 424.167,A -85,B 0,C 180,E1 -17755.409,E2 -17755.409} C_VEL
LIN {X 0,Y 275.005,Z 411.437,A -85,B 0,C 180,E1 -17760.738,E2 -17760.738} C_VEL
LIN {X 0,Y 274.54,Z 407.743,A -85,B 0,C 180,E1 -17762.352,E2 -17762.352} C_VEL
LIN {X 0,Y 272.448,Z 397.845,A -85,B 0,C 180,E1 -17766.901,E2 -17766.901} C_VEL
LIN {X 0,Y 270.65,Z 389.001,A -85,B 0,C 180,E1 -17771.145,E2 -17771.145} C_VEL
LIN {X 0,Y 270.227,Z 386.827,A -85,B 0,C 180,E1 -17772.248,E2 -17772.248} C_VEL
LIN {X 0,Y 270.173,Z 386.828,A -85,B 0,C 180,E1 -17776.749,E2 -17776.749} C_VEL
LIN {X 0,Y 270.222,Z 386.823,A -85,B 0,C 180,E1 -17781.283,E2 -17781.283} C_VEL
LIN {X 0,Y 270.215,Z 386.822,A -85,B 0,C 180,E1 -17785.096,E2 -17785.096} C_VEL
LIN {X 0,Y 270.2,Z 386.825,A -85,B 0,C 180,E1 -17789.13,E2 -17789.13} C_VEL
LIN {X 0,Y 270.264,Z 386.82,A -85,B 0,C 180,E1 -17792.146,E2 -17792.146} C_VEL
LIN {X 0,Y 270.278,Z 386.816,A -85,B 0,C 180,E1 -17795.519,E2 -17795.519} C_VEL
LIN {X 0,Y 270.302,Z 386.814,A -85,B 0,C 180,E1 -17800.244,E2 -17800.244} C_VEL
LIN {X 0,Y 270.403,Z 386.799,A -85,B 0,C 180,E1 -17804.935,E2 -17804.935} C_VEL
LIN {X 0,Y 270.442,Z 386.798,A -85,B 0,C 180,E1 -17809.519,E2 -17809.519} C_VEL
LIN {X 0,Y 270.612,Z 386.773,A -85,B 0,C 180,E1 -17812.539,E2 -17812.539} C_VEL
LIN {X 0,Y 270.791,Z 386.751,A -85,B 0,C 180,E1 -17818.513,E2 -17818.513} C_VEL
LIN {X 0,Y 270.788,Z 386.755,A -85,B 0,C 180,E1 -17821.487,E2 -17821.487} C_VEL
LIN {X 0,Y 270.612,Z 386.776,A -85,B 0,C 180,E1 -17827.461,E2 -17827.461} C_VEL
LIN {X 0,Y 270.443,Z 386.794,A -85,B 0,C 180,E1 -17830.481,E2 -17830.481} C_VEL
LIN {X 0,Y 270.404,Z 386.803,A -85,B 0,C 180,E1 -17835.065,E2 -17835.065} C_VEL
LIN {X 0,Y 270.302,Z 386.813,A -85,B 0,C 180,E1 -17839.756,E2 -17839.756} C_VEL
LIN {X 0,Y 270.275,Z 386.816,A -85,B 0,C 180,E1 -17844.586,E2 -17844.586} C_VEL
LIN {X 0,Y 270.272,Z 386.816,A -85,B 0,C 180,E1 -17847.909,E2 -17847.909} C_VEL
LIN {X 0,Y 270.185,Z 386.829,A -85,B 0,C 180,E1 -17851.348,E2 -17851.348} C_VEL
LIN {X 0,Y 270.202,Z 386.828,A -85,B 0,C 180,E1 -17854.906,E2 -17854.906} C_VEL
LIN {X 0,Y 270.198,Z 386.829,A -85,B 0,C 180,E1 -17858.711,E2 -17858.711} C_VEL
LIN {X 0,Y 270.172,Z 386.829,A -85,B 0,C 180,E1 -17863.251,E2 -17863.251} C_VEL
LIN {X 0,Y 270.175,Z 386.829,A -85,B 0,C 180,E1 -17867.443,E2 -17867.443} C_VEL
LIN {X 0,Y 270.207,Z 386.823,A -85,B 0,C 180,E1 -17871.374,E2 -17871.374} C_VEL
LIN {X 0,Y 270.216,Z 386.824,A -85,B 0,C 180,E1 -17875.097,E2 -17875.097} C_VEL
LIN {X 0,Y 270.201,Z 386.824,A -85,B 0,C 180,E1 -17879.131,E2 -17879.131} C_VEL
LIN {X 0,Y 270.264,Z 386.819,A -85,B 0,C 180,E1 -17882.147,E2 -17882.147} C_VEL
LIN {X 0,Y 270.279,Z 386.815,A -85,B 0,C 180,E1 -17885.519,E2 -17885.519} C_VEL
LIN {X 0,Y 270.305,Z 386.815,A -85,B 0,C 180,E1 -17890.245,E2 -17890.245} C_VEL
LIN {X 0,Y 270.407,Z 386.799,A -85,B 0,C 180,E1 -17894.936,E2 -17894.936} C_VEL
LIN {X 0,Y 270.444,Z 386.795,A -85,B 0,C 180,E1 -17899.519,E2 -17899.519} C_VEL
LIN {X 0,Y 270.61,Z 386.776,A -85,B 0,C 180,E1 -17902.539,E2 -17902.539} C_VEL
LIN {X 0,Y 270.79,Z 386.753,A -85,B 0,C 180,E1 -17908.513,E2 -17908.513} C_VEL
LIN {X 0,Y 270.79,Z 386.753,A -85,B 0,C 180,E1 -17911.487,E2 -17911.487} C_VEL
LIN {X 0,Y 270.601,Z 386.777,A -85,B 0,C 180,E1 -17917.462,E2 -17917.462} C_VEL
LIN {X 0,Y 270.416,Z 386.798,A -85,B 0,C 180,E1 -17920.482,E2 -17920.482} C_VEL
LIN {X 0,Y 270.406,Z 386.799,A -85,B 0,C 180,E1 -17925.065,E2 -17925.065} C_VEL
LIN {X 0,Y 270.305,Z 386.815,A -85,B 0,C 180,E1 -17929.756,E2 -17929.756} C_VEL
LIN {X 0,Y 270.277,Z 386.816,A -85,B 0,C 180,E1 -17934.586,E2 -17934.586} C_VEL
LIN {X 0,Y 270.272,Z 386.817,A -85,B 0,C 180,E1 -17937.909,E2 -17937.909} C_VEL
LIN {X 0,Y 270.186,Z 386.829,A -85,B 0,C 180,E1 -17941.348,E2 -17941.348} C_VEL
LIN {X 0,Y 270.217,Z 386.824,A -85,B 0,C 180,E1 -17944.904,E2 -17944.904} C_VEL
LIN {X 0,Y 270.225,Z 386.821,A -85,B 0,C 180,E1 -17948.717,E2 -17948.717} C_VEL
LIN {X 0,Y 270.174,Z 386.833,A -85,B 0,C 180,E1 -17953.251,E2 -17953.251} C_VEL
LIN {X 0,Y 270.177,Z 386.83,A -85,B 0,C 180,E1 -17957.442,E2 -17957.442} C_VEL
LIN {X 0,Y 270.209,Z 386.827,A -85,B 0,C 180,E1 -17961.374,E2 -17961.374} C_VEL
LIN {X 0,Y 270.256,Z 386.821,A -85,B 0,C 180,E1 -17965.102,E2 -17965.102} C_VEL
LIN {X 0,Y 270.459,Z 386.966,A -85,B 0,C 180,E1 -17968.031,E2 -17968.031} C_VEL
LIN {X 0,Y 270.595,Z 389.258,A -85,B 0,C 180,E1 -17969.708,E2 -17969.708} C_VEL
LIN {X 0,Y 270.262,Z 393.794,A -85,B 0,C 180,E1 -17972.93,E2 -17972.93} C_VEL
LIN {X 0,Y 269.733,Z 399.593,A -85,B 0,C 180,E1 -17976.994,E2 -17976.994} C_VEL
LIN {X 0,Y 269.409,Z 405.406,A -85,B 0,C 180,E1 -17980.969,E2 -17980.969} C_VEL
LIN {X 0,Y 269.077,Z 411.607,A -85,B 0,C 180,E1 -17985.107,E2 -17985.107} C_VEL
LIN {X 0,Y 268.976,Z 414.665,A -85,B 0,C 180,E1 -17987.12,E2 -17987.12} C_VEL
LIN {X 0,Y 270.105,Z 427.105,A -85,B 0,C 180,E1 -17988.176,E2 -17988.176} C_VEL
LIN {X 0,Y 270.727,Z 434.397,A -85,B 0,C 180,E1 -17988.962,E2 -17988.962} C_VEL
LIN {X 0,Y 270.224,Z 444.346,A -85,B 0,C 180,E1 -17990.267,E2 -17990.267} C_VEL
LIN {X 0,Y 269.82,Z 453.707,A -85,B 0,C 180,E1 -17991.806,E2 -17991.806} C_VEL
LIN {X 0,Y 269.522,Z 462.579,A -85,B 0,C 180,E1 -17993.637,E2 -17993.637} C_VEL
LIN {X 0,Y 269.119,Z 469.773,A -85,B 0,C 180,E1 -17995.507,E2 -17995.507} C_VEL
LIN {X 0,Y 268.847,Z 475.482,A -85,B 0,C 180,E1 -17997.378,E2 -17997.378} C_VEL
LIN {X 0,Y 268.875,Z 479.886,A -85,B 0,C 180,E1 -17999.251,E2 -17999.251} C_VEL
LIN {X 0,Y 269.168,Z 483.761,A -85,B 0,C 180,E1 -18001.496,E2 -18001.496} C_VEL
LIN {X 0,Y 269.503,Z 485.552,A -85,B 0,C 180,E1 -18002.99,E2 -18002.99} C_VEL
LIN {X 0,Y 270.008,Z 486.736,A -85,B 0,C 180,E1 -18004.479,E2 -18004.479} C_VEL
LIN {X 0,Y 270.748,Z 487.291,A -85,B 0,C 180,E1 -18005.96,E2 -18005.96} C_VEL
LIN {X 0,Y 271.674,Z 487.246,A -85,B 0,C 180,E1 -18007.432,E2 -18007.432} C_VEL
LIN {X 0,Y 272.784,Z 486.627,A -85,B 0,C 180,E1 -18008.893,E2 -18008.893} C_VEL
LIN {X 0,Y 274.132,Z 485.412,A -85,B 0,C 180,E1 -18010.338,E2 -18010.338} C_VEL
LIN {X 0,Y 276.345,Z 482.499,A -85,B 0,C 180,E1 -18012.484,E2 -18012.484} C_VEL
LIN {X 0,Y 278.938,Z 478.161,A -85,B 0,C 180,E1 -18014.593,E2 -18014.593} C_VEL
LIN {X 0,Y 281.867,Z 472.266,A -85,B 0,C 180,E1 -18016.663,E2 -18016.663} C_VEL
LIN {X 0,Y 284.701,Z 465.994,A -85,B 0,C 180,E1 -18018.345,E2 -18018.345} C_VEL
LIN {X 0,Y 285.869,Z 462.744,A -85,B 0,C 180,E1 -18019.114,E2 -18019.114} C_VEL
LIN {X 0,Y 285.886,Z 455.244,A -85,B 0,C 180,E1 -18021.223,E2 -18021.223} C_VEL
LIN {X 0,Y 284.875,Z 447.377,A -85,B 0,C 180,E1 -18023.424,E2 -18023.424} C_VEL
LIN {X 0,Y 284.629,Z 446.126,A -85,B 0,C 180,E1 -18023.788,E2 -18023.788} C_VEL
LIN {X 0,Y 283.493,Z 443.29,A -85,B 0,C 180,E1 -18024.805,E2 -18024.805} C_VEL
LIN {X 0,Y 281.685,Z 441.237,A -85,B 0,C 180,E1 -18025.874,E2 -18025.874} C_VEL
LIN {X 0,Y 276.418,Z 436.644,A -85,B 0,C 180,E1 -18028.839,E2 -18028.839} C_VEL
LIN {X 0,Y 275.568,Z 435.028,A -85,B 0,C 180,E1 -18029.579,E2 -18029.579} C_VEL
LIN {X 0,Y 274.131,Z 431.115,A -85,B 0,C 180,E1 -18031.276,E2 -18031.276} C_VEL
LIN {X 0,Y 271.913,Z 426.976,A -85,B 0,C 180,E1 -18033.735,E2 -18033.735} C_VEL
LIN {X 0,Y 271.632,Z 426.02,A -85,B 0,C 180,E1 -18034.234,E2 -18034.234} C_VEL
LIN {X 0,Y 272.016,Z 425.574,A -85,B 0,C 180,E1 -18036.779,E2 -18036.779} C_VEL
LIN {X 0,Y 272.384,Z 425.673,A -85,B 0,C 180,E1 -18040.169,E2 -18040.169} C_VEL
LIN {X 0,Y 272.888,Z 426.584,A -85,B 0,C 180,E1 -18043.853,E2 -18043.853} C_VEL
LIN {X 0,Y 273.166,Z 427.624,A -85,B 0,C 180,E1 -18046.086,E2 -18046.086} C_VEL
LIN {X 0,Y 273.496,Z 428.906,A -85,B 0,C 180,E1 -18048.177,E2 -18048.177} C_VEL
LIN {X 0,Y 274.174,Z 432.113,A -85,B 0,C 180,E1 -18051.983,E2 -18051.983} C_VEL
LIN {X 0,Y 277.109,Z 437.71,A -85,B 0,C 180,E1 -18054.251,E2 -18054.251} C_VEL
LIN {X 0,Y 278.027,Z 438.934,A -85,B 0,C 180,E1 -18054.821,E2 -18054.821} C_VEL
LIN {X 0,Y 279.769,Z 443.934,A -85,B 0,C 180,E1 -18056.184,E2 -18056.184} C_VEL
LIN {X 0,Y 281.094,Z 454.982,A -85,B 0,C 180,E1 -18058.328,E2 -18058.328} C_VEL
LIN {X 0,Y 281.394,Z 466.911,A -85,B 0,C 180,E1 -18060.485,E2 -18060.485} C_VEL
LIN {X 0,Y 280.714,Z 475.901,A -85,B 0,C 180,E1 -18062.09,E2 -18062.09} C_VEL
LIN {X 0,Y 279.269,Z 483.7,A -85,B 0,C 180,E1 -18063.468,E2 -18063.468} C_VEL
LIN {X 0,Y 276.326,Z 492.929,A -85,B 0,C 180,E1 -18065.187,E2 -18065.187} C_VEL
LIN {X 0,Y 272.496,Z 502.228,A -85,B 0,C 180,E1 -18067.24,E2 -18067.24} C_VEL
LIN {X 0,Y 269.46,Z 509.856,A -85,B 0,C 180,E1 -18069.384,E2 -18069.384} C_VEL
LIN {X 0,Y 266.76,Z 516.159,A -85,B 0,C 180,E1 -18071.569,E2 -18071.569} C_VEL
LIN {X 0,Y 264.745,Z 521.255,A -85,B 0,C 180,E1 -18073.815,E2 -18073.815} C_VEL
LIN {X 0,Y 262.772,Z 526.466,A -85,B 0,C 180,E1 -18076.859,E2 -18076.859} C_VEL
LIN {X 0,Y 261.893,Z 529.266,A -85,B 0,C 180,E1 -18079.172,E2 -18079.172} C_VEL
LIN {X 0,Y 261.528,Z 531.606,A -85,B 0,C 180,E1 -18082.278,E2 -18082.278} C_VEL
LIN {X 0,Y 261.572,Z 532.203,A -85,B 0,C 180,E1 -18083.83,E2 -18083.83} C_VEL
LIN {X 0,Y 261.625,Z 532.382,A -85,B 0,C 180,E1 -18085.377,E2 -18085.377} C_VEL
LIN {X 0,Y 261.896,Z 532.138,A -85,B 0,C 180,E1 -18086.923,E2 -18086.923} C_VEL
LIN {X 0,Y 262.206,Z 531.492,A -85,B 0,C 180,E1 -18088.464,E2 -18088.464} C_VEL
LIN {X 0,Y 262.321,Z 530.37,A -85,B 0,C 180,E1 -18090,E2 -18090} C_VEL
LIN {X 0,Y 262.437,Z 527.747,A -85,B 0,C 180,E1 -18092.302,E2 -18092.302} C_VEL
LIN {X 0,Y 262.38,Z 523.899,A -85,B 0,C 180,E1 -18094.609,E2 -18094.609} C_VEL
LIN {X 0,Y 262.365,Z 518.37,A -85,B 0,C 180,E1 -18097.06,E2 -18097.06} C_VEL
LIN {X 0,Y 262.382,Z 511.957,A -85,B 0,C 180,E1 -18099.248,E2 -18099.248} C_VEL
LIN {X 0,Y 262.757,Z 503.346,A -85,B 0,C 180,E1 -18101.572,E2 -18101.572} C_VEL
LIN {X 0,Y 263.266,Z 494.311,A -85,B 0,C 180,E1 -18103.508,E2 -18103.508} C_VEL
LIN {X 0,Y 264.054,Z 484.305,A -85,B 0,C 180,E1 -18105.238,E2 -18105.238} C_VEL
LIN {X 0,Y 264.718,Z 474.643,A -85,B 0,C 180,E1 -18106.583,E2 -18106.583} C_VEL
LIN {X 0,Y 264.253,Z 465.672,A -85,B 0,C 180,E1 -18107.589,E2 -18107.589} C_VEL
LIN {X 0,Y 263.408,Z 452.012,A -85,B 0,C 180,E1 -18108.774,E2 -18108.774} C_VEL
LIN {X 0,Y 263.06,Z 439.974,A -85,B 0,C 180,E1 -18109.509,E2 -18109.509} C_VEL
LIN {X 0,Y 263.113,Z 437.942,A -85,B 0,C 180,E1 -18109.606,E2 -18109.606} C_VEL
LIN {X 0,Y 265.088,Z 425.284,A -85,B 0,C 180,E1 -18115.099,E2 -18115.099} C_VEL
LIN {X 0,Y 267.901,Z 412.188,A -85,B 0,C 180,E1 -18120.767,E2 -18120.767} C_VEL
LIN {X 0,Y 267.573,Z 409.032,A -85,B 0,C 180,E1 -18122.189,E2 -18122.189} C_VEL
LIN {X 0,Y 265.613,Z 399.923,A -85,B 0,C 180,E1 -18126.446,E2 -18126.446} C_VEL
LIN {X 0,Y 264.077,Z 392.378,A -85,B 0,C 180,E1 -18130.169,E2 -18130.169} C_VEL
LIN {X 0,Y 263.204,Z 387.702,A -85,B 0,C 180,E1 -18132.564,E2 -18132.564} C_VEL
LIN {X 0,Y 263.13,Z 387.709,A -85,B 0,C 180,E1 -18136.149,E2 -18136.149} C_VEL
LIN {X 0,Y 263.116,Z 387.712,A -85,B 0,C 180,E1 -18140.129,E2 -18140.129} C_VEL
LIN {X 0,Y 263.188,Z 387.702,A -85,B 0,C 180,E1 -18144.022,E2 -18144.022} C_VEL
LIN {X 0,Y 263.134,Z 387.707,A -85,B 0,C 180,E1 -18147.712,E2 -18147.712} C_VEL
LIN {X 0,Y 263.196,Z 387.701,A -85,B 0,C 180,E1 -18151.785,E2 -18151.785} C_VEL
LIN {X 0,Y 263.226,Z 387.693,A -85,B 0,C 180,E1 -18155.2,E2 -18155.2} C_VEL
LIN {X 0,Y 263.264,Z 387.693,A -85,B 0,C 180,E1 -18159.693,E2 -18159.693} C_VEL
LIN {X 0,Y 263.352,Z 387.678,A -85,B 0,C 180,E1 -18164.522,E2 -18164.522} C_VEL
LIN {X 0,Y 263.375,Z 387.677,A -85,B 0,C 180,E1 -18169.234,E2 -18169.234} C_VEL
LIN {X 0,Y 263.574,Z 387.65,A -85,B 0,C 180,E1 -18172.338,E2 -18172.338} C_VEL
LIN {X 0,Y 263.755,Z 387.627,A -85,B 0,C 180,E1 -18178.473,E2 -18178.473} C_VEL
LIN {X 0,Y 263.752,Z 387.632,A -85,B 0,C 180,E1 -18181.527,E2 -18181.527} C_VEL
LIN {X 0,Y 263.574,Z 387.651,A -85,B 0,C 180,E1 -18187.662,E2 -18187.662} C_VEL
LIN {X 0,Y 263.376,Z 387.676,A -85,B 0,C 180,E1 -18190.766,E2 -18190.766} C_VEL
LIN {X 0,Y 263.352,Z 387.68,A -85,B 0,C 180,E1 -18195.478,E2 -18195.478} C_VEL
LIN {X 0,Y 263.264,Z 387.689,A -85,B 0,C 180,E1 -18200.307,E2 -18200.307} C_VEL
LIN {X 0,Y 263.209,Z 387.697,A -85,B 0,C 180,E1 -18205.291,E2 -18205.291} C_VEL
LIN {X 0,Y 263.18,Z 387.702,A -85,B 0,C 180,E1 -18208.73,E2 -18208.73} C_VEL
LIN {X 0,Y 263.134,Z 387.706,A -85,B 0,C 180,E1 -18212.288,E2 -18212.288} C_VEL
LIN {X 0,Y 263.183,Z 387.702,A -85,B 0,C 180,E1 -18216.764,E2 -18216.764} C_VEL
LIN {X 0,Y 263.125,Z 387.705,A -85,B 0,C 180,E1 -18221.594,E2 -18221.594} C_VEL
LIN {X 0,Y 263.128,Z 387.706,A -85,B 0,C 180,E1 -18226.017,E2 -18226.017} C_VEL
LIN {X 0,Y 263.116,Z 387.708,A -85,B 0,C 180,E1 -18230.13,E2 -18230.13} C_VEL
LIN {X 0,Y 263.189,Z 387.699,A -85,B 0,C 180,E1 -18234.022,E2 -18234.022} C_VEL
LIN {X 0,Y 263.134,Z 387.705,A -85,B 0,C 180,E1 -18237.712,E2 -18237.712} C_VEL
LIN {X 0,Y 263.199,Z 387.697,A -85,B 0,C 180,E1 -18241.785,E2 -18241.785} C_VEL
LIN {X 0,Y 263.227,Z 387.694,A -85,B 0,C 180,E1 -18245.201,E2 -18245.201} C_VEL
LIN {X 0,Y 263.271,Z 387.688,A -85,B 0,C 180,E1 -18249.694,E2 -18249.694} C_VEL
LIN {X 0,Y 263.354,Z 387.68,A -85,B 0,C 180,E1 -18254.522,E2 -18254.522} C_VEL
LIN {X 0,Y 263.376,Z 387.675,A -85,B 0,C 180,E1 -18259.235,E2 -18259.235} C_VEL
LIN {X 0,Y 263.572,Z 387.654,A -85,B 0,C 180,E1 -18262.339,E2 -18262.339} C_VEL
LIN {X 0,Y 263.754,Z 387.63,A -85,B 0,C 180,E1 -18268.473,E2 -18268.473} C_VEL
LIN {X 0,Y 263.754,Z 387.63,A -85,B 0,C 180,E1 -18271.527,E2 -18271.527} C_VEL
LIN {X 0,Y 263.561,Z 387.655,A -85,B 0,C 180,E1 -18277.662,E2 -18277.662} C_VEL
LIN {X 0,Y 263.358,Z 387.677,A -85,B 0,C 180,E1 -18280.767,E2 -18280.767} C_VEL
LIN {X 0,Y 263.354,Z 387.68,A -85,B 0,C 180,E1 -18285.478,E2 -18285.478} C_VEL
LIN {X 0,Y 263.267,Z 387.688,A -85,B 0,C 180,E1 -18290.307,E2 -18290.307} C_VEL
LIN {X 0,Y 263.211,Z 387.698,A -85,B 0,C 180,E1 -18295.291,E2 -18295.291} C_VEL
LIN {X 0,Y 263.178,Z 387.699,A -85,B 0,C 180,E1 -18298.73,E2 -18298.73} C_VEL
LIN {X 0,Y 263.136,Z 387.705,A -85,B 0,C 180,E1 -18302.288,E2 -18302.288} C_VEL
LIN {X 0,Y 263.19,Z 387.699,A -85,B 0,C 180,E1 -18305.978,E2 -18305.978} C_VEL
LIN {X 0,Y 263.118,Z 387.708,A -85,B 0,C 180,E1 -18309.871,E2 -18309.871} C_VEL
LIN {X 0,Y 263.13,Z 387.706,A -85,B 0,C 180,E1 -18313.983,E2 -18313.983} C_VEL
LIN {X 0,Y 263.127,Z 387.705,A -85,B 0,C 180,E1 -18318.406,E2 -18318.406} C_VEL
LIN {X 0,Y 263.192,Z 387.701,A -85,B 0,C 180,E1 -18323.235,E2 -18323.235} C_VEL
LIN {X 0,Y 263.43,Z 387.862,A -85,B 0,C 180,E1 -18328.01,E2 -18328.01} C_VEL
LIN {X 0,Y 263.504,Z 391.114,A -85,B 0,C 180,E1 -18330.434,E2 -18330.434} C_VEL
LIN {X 0,Y 262.944,Z 397.015,A -85,B 0,C 180,E1 -18334.681,E2 -18334.681} C_VEL
LIN {X 0,Y 262.466,Z 404.048,A -85,B 0,C 180,E1 -18339.629,E2 -18339.629} C_VEL
LIN {X 0,Y 262.048,Z 411.101,A -85,B 0,C 180,E1 -18344.443,E2 -18344.443} C_VEL
LIN {X 0,Y 261.89,Z 415.005,A -85,B 0,C 180,E1 -18347.061,E2 -18347.061} C_VEL
LIN {X 0,Y 263.103,Z 428.221,A -85,B 0,C 180,E1 -18348.248,E2 -18348.248} C_VEL
LIN {X 0,Y 263.645,Z 433.761,A -85,B 0,C 180,E1 -18348.857,E2 -18348.857} C_VEL
LIN {X 0,Y 263.148,Z 443.972,A -85,B 0,C 180,E1 -18350.197,E2 -18350.197} C_VEL
LIN {X 0,Y 262.686,Z 454.323,A -85,B 0,C 180,E1 -18351.925,E2 -18351.925} C_VEL
LIN {X 0,Y 262.399,Z 463.405,A -85,B 0,C 180,E1 -18353.85,E2 -18353.85} C_VEL
LIN {X 0,Y 261.972,Z 470.506,A -85,B 0,C 180,E1 -18355.769,E2 -18355.769} C_VEL
LIN {X 0,Y 261.752,Z 476.191,A -85,B 0,C 180,E1 -18357.692,E2 -18357.692} C_VEL
LIN {X 0,Y 261.832,Z 481.404,A -85,B 0,C 180,E1 -18360,E2 -18360} C_VEL
LIN {X 0,Y 262.076,Z 484.013,A -85,B 0,C 180,E1 -18361.537,E2 -18361.537} C_VEL
LIN {X 0,Y 262.449,Z 485.955,A -85,B 0,C 180,E1 -18363.07,E2 -18363.07} C_VEL
LIN {X 0,Y 262.964,Z 487.295,A -85,B 0,C 180,E1 -18364.599,E2 -18364.599} C_VEL
LIN {X 0,Y 263.748,Z 488.05,A -85,B 0,C 180,E1 -18366.119,E2 -18366.119} C_VEL
LIN {X 0,Y 264.701,Z 488.219,A -85,B 0,C 180,E1 -18367.629,E2 -18367.629} C_VEL
LIN {X 0,Y 265.863,Z 487.782,A -85,B 0,C 180,E1 -18369.126,E2 -18369.126} C_VEL
LIN {X 0,Y 267.273,Z 486.767,A -85,B 0,C 180,E1 -18370.607,E2 -18370.607} C_VEL
LIN {X 0,Y 269.602,Z 484.185,A -85,B 0,C 180,E1 -18372.802,E2 -18372.802} C_VEL
LIN {X 0,Y 272.324,Z 480.221,A -85,B 0,C 180,E1 -18374.956,E2 -18374.956} C_VEL
LIN {X 0,Y 275.404,Z 474.811,A -85,B 0,C 180,E1 -18377.066,E2 -18377.066} C_VEL
LIN {X 0,Y 278.935,Z 467.613,A -85,B 0,C 180,E1 -18379.12,E2 -18379.12} C_VEL
LIN {X 0,Y 279.925,Z 465.091,A -85,B 0,C 180,E1 -18379.761,E2 -18379.761} C_VEL
LIN {X 0,Y 280.188,Z 457.399,A -85,B 0,C 180,E1 -18382.101,E2 -18382.101} C_VEL
LIN {X 0,Y 279.385,Z 449.888,A -85,B 0,C 180,E1 -18384.415,E2 -18384.415} C_VEL
LIN {X 0,Y 278.042,Z 443.135,A -85,B 0,C 180,E1 -18386.599,E2 -18386.599} C_VEL
LIN {X 0,Y 276.776,Z 438.652,A -85,B 0,C 180,E1 -18388.171,E2 -18388.171} C_VEL
LIN {X 0,Y 275.568,Z 435.028,A -85,B 0,C 180,E1 -18389.579,E2 -18389.579} C_VEL
LIN {X 0,Y 274.262,Z 433.057,A -85,B 0,C 180,E1 -18390.703,E2 -18390.703} C_VEL
LIN {X 0,Y 272.547,Z 432.177,A -85,B 0,C 180,E1 -18391.881,E2 -18391.881} C_VEL
LIN {X 0,Y 268.112,Z 431.701,A -85,B 0,C 180,E1 -18395.17,E2 -18395.17} C_VEL
LIN {X 0,Y 267.445,Z 431.241,A -85,B 0,C 180,E1 -18396.018,E2 -18396.018} C_VEL
LIN {X 0,Y 265.996,Z 428.757,A -85,B 0,C 180,E1 -18399.983,E2 -18399.983} C_VEL
LIN {X 0,Y 265.947,Z 428.491,A -85,B 0,C 180,E1 -18401.35,E2 -18401.35} C_VEL
LIN {X 0,Y 266.419,Z 429.779,A -85,B 0,C 180,E1 -18405.045,E2 -18405.045} C_VEL
LIN {X 0,Y 267.936,Z 433.432,A -85,B 0,C 180,E1 -18408.285,E2 -18408.285} C_VEL
LIN {X 0,Y 271.051,Z 438.139,A -85,B 0,C 180,E1 -18411.516,E2 -18411.516} C_VEL
LIN {X 0,Y 273.548,Z 443.444,A -85,B 0,C 180,E1 -18413.777,E2 -18413.777} C_VEL
LIN {X 0,Y 274.402,Z 444.693,A -85,B 0,C 180,E1 -18414.361,E2 -18414.361} C_VEL
LIN {X 0,Y 275.559,Z 448.96,A -85,B 0,C 180,E1 -18415.583,E2 -18415.583} C_VEL
LIN {X 0,Y 276.186,Z 459.188,A -85,B 0,C 180,E1 -18417.698,E2 -18417.698} C_VEL
LIN {X 0,Y 275.951,Z 469.616,A -85,B 0,C 180,E1 -18419.728,E2 -18419.728} C_VEL
LIN {X 0,Y 274.752,Z 479.552,A -85,B 0,C 180,E1 -18421.623,E2 -18421.623} C_VEL
LIN {X 0,Y 272.609,Z 487.676,A -85,B 0,C 180,E1 -18423.182,E2 -18423.182} C_VEL
LIN {X 0,Y 269.347,Z 496.167,A -85,B 0,C 180,E1 -18424.912,E2 -18424.912} C_VEL
LIN {X 0,Y 265.415,Z 504.688,A -85,B 0,C 180,E1 -18427.01,E2 -18427.01} C_VEL
LIN {X 0,Y 262.32,Z 511.645,A -85,B 0,C 180,E1 -18429.207,E2 -18429.207} C_VEL
LIN {X 0,Y 259.525,Z 517.745,A -85,B 0,C 180,E1 -18431.606,E2 -18431.606} C_VEL
LIN {X 0,Y 257.343,Z 522.724,A -85,B 0,C 180,E1 -18434.151,E2 -18434.151} C_VEL
LIN {X 0,Y 255.402,Z 527.209,A -85,B 0,C 180,E1 -18437.282,E2 -18437.282} C_VEL
LIN {X 0,Y 254.572,Z 530.064,A -85,B 0,C 180,E1 -18440.465,E2 -18440.465} C_VEL
LIN {X 0,Y 254.479,Z 530.944,A -85,B 0,C 180,E1 -18442.063,E2 -18442.063} C_VEL
LIN {X 0,Y 254.528,Z 531.411,A -85,B 0,C 180,E1 -18443.737,E2 -18443.737} C_VEL
LIN {X 0,Y 254.871,Z 531.123,A -85,B 0,C 180,E1 -18446.838,E2 -18446.838} C_VEL
LIN {X 0,Y 255.183,Z 530.36,A -85,B 0,C 180,E1 -18448.422,E2 -18448.422} C_VEL
LIN {X 0,Y 255.331,Z 529.097,A -85,B 0,C 180,E1 -18450,E2 -18450} C_VEL
LIN {X 0,Y 255.462,Z 526.3,A -85,B 0,C 180,E1 -18452.365,E2 -18452.365} C_VEL
LIN {X 0,Y 255.39,Z 522.247,A -85,B 0,C 180,E1 -18454.735,E2 -18454.735} C_VEL
LIN {X 0,Y 255.371,Z 516.53,A -85,B 0,C 180,E1 -18457.217,E2 -18457.217} C_VEL
LIN {X 0,Y 255.41,Z 509.724,A -85,B 0,C 180,E1 -18459.503,E2 -18459.503} C_VEL
LIN {X 0,Y 255.751,Z 502.418,A -85,B 0,C 180,E1 -18461.492,E2 -18461.492} C_VEL
LIN {X 0,Y 256.239,Z 493.333,A -85,B 0,C 180,E1 -18463.481,E2 -18463.481} C_VEL
LIN {X 0,Y 257.02,Z 483.279,A -85,B 0,C 180,E1 -18465.259,E2 -18465.259} C_VEL
LIN {X 0,Y 257.645,Z 473.775,A -85,B 0,C 180,E1 -18466.605,E2 -18466.605} C_VEL
LIN {X 0,Y 257.005,Z 462.995,A -85,B 0,C 180,E1 -18467.814,E2 -18467.814} C_VEL
LIN {X 0,Y 256.243,Z 450.37,A -85,B 0,C 180,E1 -18468.904,E2 -18468.904} C_VEL
LIN {X 0,Y 255.999,Z 439.032,A -85,B 0,C 180,E1 -18469.599,E2 -18469.599} C_VEL
LIN {X 0,Y 256.084,Z 437.455,A -85,B 0,C 180,E1 -18469.749,E2 -18469.749} C_VEL
LIN {X 0,Y 258.246,Z 424.01,A -85,B 0,C 180,E1 -18475.812,E2 -18475.812} C_VEL
LIN {X 0,Y 260.774,Z 412.832,A -85,B 0,C 180,E1 -18480.801,E2 -18480.801} C_VEL
LIN {X 0,Y 260.525,Z 409.818,A -85,B 0,C 180,E1 -18482.193,E2 -18482.193} C_VEL
LIN {X 0,Y 258.487,Z 400.467,A -85,B 0,C 180,E1 -18486.738,E2 -18486.738} C_VEL
LIN {X 0,Y 257.146,Z 393.859,A -85,B 0,C 180,E1 -18490.07,E2 -18490.07} C_VEL
LIN {X 0,Y 256.146,Z 388.58,A -85,B 0,C 180,E1 -18492.915,E2 -18492.915} C_VEL
LIN {X 0,Y 256.074,Z 388.584,A -85,B 0,C 180,E1 -18497.818,E2 -18497.818} C_VEL
LIN {X 0,Y 256.089,Z 388.584,A -85,B 0,C 180,E1 -18500.861,E2 -18500.861} C_VEL
LIN {X 0,Y 256.121,Z 388.578,A -85,B 0,C 180,E1 -18504.813,E2 -18504.813} C_VEL
LIN {X 0,Y 256.093,Z 388.583,A -85,B 0,C 180,E1 -18508.572,E2 -18508.572} C_VEL
LIN {X 0,Y 256.138,Z 388.579,A -85,B 0,C 180,E1 -18512.196,E2 -18512.196} C_VEL
LIN {X 0,Y 256.168,Z 388.574,A -85,B 0,C 180,E1 -18515.699,E2 -18515.699} C_VEL
LIN {X 0,Y 256.167,Z 388.574,A -85,B 0,C 180,E1 -18519.105,E2 -18519.105} C_VEL
LIN {X 0,Y 256.301,Z 388.558,A -85,B 0,C 180,E1 -18524.085,E2 -18524.085} C_VEL
LIN {X 0,Y 256.31,Z 388.556,A -85,B 0,C 180,E1 -18528.934,E2 -18528.934} C_VEL
LIN {X 0,Y 256.541,Z 388.527,A -85,B 0,C 180,E1 -18532.127,E2 -18532.127} C_VEL
LIN {X 0,Y 256.718,Z 388.504,A -85,B 0,C 180,E1 -18538.431,E2 -18538.431} C_VEL
LIN {X 0,Y 256.715,Z 388.509,A -85,B 0,C 180,E1 -18541.569,E2 -18541.569} C_VEL
LIN {X 0,Y 256.541,Z 388.526,A -85,B 0,C 180,E1 -18547.873,E2 -18547.873} C_VEL
LIN {X 0,Y 256.311,Z 388.557,A -85,B 0,C 180,E1 -18551.066,E2 -18551.066} C_VEL
LIN {X 0,Y 256.301,Z 388.556,A -85,B 0,C 180,E1 -18555.915,E2 -18555.915} C_VEL
LIN {X 0,Y 256.168,Z 388.576,A -85,B 0,C 180,E1 -18560.895,E2 -18560.895} C_VEL
LIN {X 0,Y 256.189,Z 388.572,A -85,B 0,C 180,E1 -18565.139,E2 -18565.139} C_VEL
LIN {X 0,Y 256.114,Z 388.581,A -85,B 0,C 180,E1 -18569.6,E2 -18569.6} C_VEL
LIN {X 0,Y 256.068,Z 388.586,A -85,B 0,C 180,E1 -18573.293,E2 -18573.293} C_VEL
LIN {X 0,Y 256.115,Z 388.582,A -85,B 0,C 180,E1 -18577.271,E2 -18577.271} C_VEL
LIN {X 0,Y 256.056,Z 388.588,A -85,B 0,C 180,E1 -18581.203,E2 -18581.203} C_VEL
LIN {X 0,Y 256.063,Z 388.586,A -85,B 0,C 180,E1 -18585.529,E2 -18585.529} C_VEL
LIN {X 0,Y 256.058,Z 388.59,A -85,B 0,C 180,E1 -18588.798,E2 -18588.798} C_VEL
LIN {X 0,Y 256.146,Z 388.578,A -85,B 0,C 180,E1 -18592.87,E2 -18592.87} C_VEL
LIN {X 0,Y 256.086,Z 388.586,A -85,B 0,C 180,E1 -18596.71,E2 -18596.71} C_VEL
LIN {X 0,Y 256.135,Z 388.576,A -85,B 0,C 180,E1 -18601.407,E2 -18601.407} C_VEL
LIN {X 0,Y 256.17,Z 388.573,A -85,B 0,C 180,E1 -18605.7,E2 -18605.7} C_VEL
LIN {X 0,Y 256.22,Z 388.565,A -85,B 0,C 180,E1 -18609.11,E2 -18609.11} C_VEL
LIN {X 0,Y 256.303,Z 388.56,A -85,B 0,C 180,E1 -18614.086,E2 -18614.086} C_VEL
LIN {X 0,Y 256.312,Z 388.555,A -85,B 0,C 180,E1 -18618.934,E2 -18618.934} C_VEL
LIN {X 0,Y 256.54,Z 388.531,A -85,B 0,C 180,E1 -18622.127,E2 -18622.127} C_VEL
LIN {X 0,Y 256.717,Z 388.506,A -85,B 0,C 180,E1 -18628.432,E2 -18628.432} C_VEL
LIN {X 0,Y 256.717,Z 388.506,A -85,B 0,C 180,E1 -18631.569,E2 -18631.569} C_VEL
LIN {X 0,Y 256.484,Z 388.535,A -85,B 0,C 180,E1 -18636.293,E2 -18636.293} C_VEL
LIN {X 0,Y 256.429,Z 388.543,A -85,B 0,C 180,E1 -18639.465,E2 -18639.465} C_VEL
LIN {X 0,Y 256.258,Z 388.562,A -85,B 0,C 180,E1 -18644.29,E2 -18644.29} C_VEL
LIN {X 0,Y 256.214,Z 388.571,A -85,B 0,C 180,E1 -18647.562,E2 -18647.562} C_VEL
LIN {X 0,Y 256.162,Z 388.573,A -85,B 0,C 180,E1 -18651.121,E2 -18651.121} C_VEL
LIN {X 0,Y 256.191,Z 388.572,A -85,B 0,C 180,E1 -18655.139,E2 -18655.139} C_VEL
LIN {X 0,Y 256.113,Z 388.582,A -85,B 0,C 180,E1 -18659.6,E2 -18659.6} C_VEL
LIN {X 0,Y 256.088,Z 388.586,A -85,B 0,C 180,E1 -18663.29,E2 -18663.29} C_VEL
LIN {X 0,Y 256.131,Z 388.581,A -85,B 0,C 180,E1 -18667.275,E2 -18667.275} C_VEL
LIN {X 0,Y 256.06,Z 388.59,A -85,B 0,C 180,E1 -18671.203,E2 -18671.203} C_VEL
LIN {X 0,Y 256.065,Z 388.587,A -85,B 0,C 180,E1 -18675.529,E2 -18675.529} C_VEL
LIN {X 0,Y 256.058,Z 388.587,A -85,B 0,C 180,E1 -18678.797,E2 -18678.797} C_VEL
LIN {X 0,Y 256.138,Z 388.58,A -85,B 0,C 180,E1 -18682.869,E2 -18682.869} C_VEL
LIN {X 0,Y 256.36,Z 388.631,A -85,B 0,C 180,E1 -18687.911,E2 -18687.911} C_VEL
LIN {X 0,Y 256.492,Z 390.769,A -85,B 0,C 180,E1 -18689.542,E2 -18689.542} C_VEL
LIN {X 0,Y 256.099,Z 395.562,A -85,B 0,C 180,E1 -18693.076,E2 -18693.076} C_VEL
LIN {X 0,Y 255.555,Z 401.455,A -85,B 0,C 180,E1 -18697.355,E2 -18697.355} C_VEL
LIN {X 0,Y 255.193,Z 407.362,A -85,B 0,C 180,E1 -18701.536,E2 -18701.536} C_VEL
LIN {X 0,Y 254.876,Z 413.256,A -85,B 0,C 180,E1 -18705.631,E2 -18705.631} C_VEL
LIN {X 0,Y 254.828,Z 415.382,A -85,B 0,C 180,E1 -18707.051,E2 -18707.051} C_VEL
LIN {X 0,Y 255.855,Z 427.323,A -85,B 0,C 180,E1 -18708.111,E2 -18708.111} C_VEL
LIN {X 0,Y 256.518,Z 434.77,A -85,B 0,C 180,E1 -18708.943,E2 -18708.943} C_VEL
LIN {X 0,Y 255.965,Z 446.109,A -85,B 0,C 180,E1 -18710.518,E2 -18710.518} C_VEL
LIN {X 0,Y 255.526,Z 455.051,A -85,B 0,C 180,E1 -18712.096,E2 -18712.096} C_VEL
LIN {X 0,Y 255.3,Z 464.047,A -85,B 0,C 180,E1 -18714.075,E2 -18714.075} C_VEL
LIN {X 0,Y 254.84,Z 471.176,A -85,B 0,C 180,E1 -18716.047,E2 -18716.047} C_VEL
LIN {X 0,Y 254.642,Z 476.898,A -85,B 0,C 180,E1 -18718.023,E2 -18718.023} C_VEL
LIN {X 0,Y 254.731,Z 481.344,A -85,B 0,C 180,E1 -18720,E2 -18720} C_VEL
LIN {X 0,Y 255.177,Z 485.275,A -85,B 0,C 180,E1 -18722.368,E2 -18722.368} C_VEL
LIN {X 0,Y 255.923,Z 487.83,A -85,B 0,C 180,E1 -18724.726,E2 -18724.726} C_VEL
LIN {X 0,Y 256.75,Z 488.761,A -85,B 0,C 180,E1 -18726.286,E2 -18726.286} C_VEL
LIN {X 0,Y 257.722,Z 489.109,A -85,B 0,C 180,E1 -18727.837,E2 -18727.837} C_VEL
LIN {X 0,Y 258.94,Z 488.896,A -85,B 0,C 180,E1 -18729.372,E2 -18729.372} C_VEL
LIN {X 0,Y 260.416,Z 488.097,A -85,B 0,C 180,E1 -18730.889,E2 -18730.889} C_VEL
LIN {X 0,Y 261.992,Z 486.712,A -85,B 0,C 180,E1 -18732.392,E2 -18732.392} C_VEL
LIN {X 0,Y 264.712,Z 483.596,A -85,B 0,C 180,E1 -18734.609,E2 -18734.609} C_VEL
LIN {X 0,Y 267.827,Z 479.078,A -85,B 0,C 180,E1 -18736.777,E2 -18736.777} C_VEL
LIN {X 0,Y 271.33,Z 473.044,A -85,B 0,C 180,E1 -18738.891,E2 -18738.891} C_VEL
LIN {X 0,Y 273.867,Z 468.067,A -85,B 0,C 180,E1 -18740.27,E2 -18740.27} C_VEL
LIN {X 0,Y 274.522,Z 461.749,A -85,B 0,C 180,E1 -18742.345,E2 -18742.345} C_VEL
LIN {X 0,Y 274.367,Z 456.181,A -85,B 0,C 180,E1 -18744.195,E2 -18744.195} C_VEL
LIN {X 0,Y 273.496,Z 449.141,A -85,B 0,C 180,E1 -18746.63,E2 -18746.63} C_VEL
LIN {X 0,Y 272.388,Z 443.682,A -85,B 0,C 180,E1 -18748.687,E2 -18748.687} C_VEL
LIN {X 0,Y 271.336,Z 439.883,A -85,B 0,C 180,E1 -18750.289,E2 -18750.289} C_VEL
LIN {X 0,Y 270.364,Z 436.773,A -85,B 0,C 180,E1 -18751.762,E2 -18751.762} C_VEL
LIN {X 0,Y 268.672,Z 432.904,A -85,B 0,C 180,E1 -18754.198,E2 -18754.198} C_VEL
LIN {X 0,Y 267.445,Z 431.241,A -85,B 0,C 180,E1 -18756.018,E2 -18756.018} C_VEL
LIN {X 0,Y 266.544,Z 430.948,A -85,B 0,C 180,E1 -18757.269,E2 -18757.269} C_VEL
LIN {X 0,Y 264.804,Z 432.427,A -85,B 0,C 180,E1 -18759.349,E2 -18759.349} C_VEL
LIN {X 0,Y 263.385,Z 434.977,A -85,B 0,C 180,E1 -18761.887,E2 -18761.887} C_VEL
LIN {X 0,Y 263.324,Z 435.448,A -85,B 0,C 180,E1 -18762.753,E2 -18762.753} C_VEL
LIN {X 0,Y 263.501,Z 435.825,A -85,B 0,C 180,E1 -18763.934,E2 -18763.934} C_VEL
LIN {X 0,Y 264.196,Z 437.672,A -85,B 0,C 180,E1 -18766.24,E2 -18766.24} C_VEL
LIN {X 0,Y 266.489,Z 442.381,A -85,B 0,C 180,E1 -18769.89,E2 -18769.89} C_VEL
LIN {X 0,Y 267.452,Z 443.818,A -85,B 0,C 180,E1 -18770.901,E2 -18770.901} C_VEL
LIN {X 0,Y 270.26,Z 449.858,A -85,B 0,C 180,E1 -18773.721,E2 -18773.721} C_VEL
LIN {X 0,Y 271.169,Z 453.085,A -85,B 0,C 180,E1 -18774.8,E2 -18774.8} C_VEL
LIN {X 0,Y 271.233,Z 463.218,A -85,B 0,C 180,E1 -18777.034,E2 -18777.034} C_VEL
LIN {X 0,Y 270.339,Z 474.315,A -85,B 0,C 180,E1 -18779.352,E2 -18779.352} C_VEL
LIN {X 0,Y 268.758,Z 482.628,A -85,B 0,C 180,E1 -18781.067,E2 -18781.067} C_VEL
LIN {X 0,Y 265.881,Z 491.421,A -85,B 0,C 180,E1 -18782.872,E2 -18782.872} C_VEL
LIN {X 0,Y 261.653,Z 500.49,A -85,B 0,C 180,E1 -18784.973,E2 -18784.973} C_VEL
LIN {X 0,Y 258.502,Z 506.882,A -85,B 0,C 180,E1 -18786.782,E2 -18786.782} C_VEL
LIN {X 0,Y 255.211,Z 513.291,A -85,B 0,C 180,E1 -18789.023,E2 -18789.023} C_VEL
LIN {X 0,Y 252.674,Z 518.263,A -85,B 0,C 180,E1 -18791.216,E2 -18791.216} C_VEL
LIN {X 0,Y 250.477,Z 522.73,A -85,B 0,C 180,E1 -18793.705,E2 -18793.705} C_VEL
LIN {X 0,Y 249.413,Z 525.002,A -85,B 0,C 180,E1 -18795.309,E2 -18795.309} C_VEL
LIN {X 0,Y 248.452,Z 526.864,A -85,B 0,C 180,E1 -18796.92,E2 -18796.92} C_VEL
LIN {X 0,Y 247.534,Z 529.483,A -85,B 0,C 180,E1 -18800.191,E2 -18800.191} C_VEL
LIN {X 0,Y 247.454,Z 530.544,A -85,B 0,C 180,E1 -18803.476,E2 -18803.476} C_VEL
LIN {X 0,Y 247.524,Z 530.498,A -85,B 0,C 180,E1 -18805.113,E2 -18805.113} C_VEL
LIN {X 0,Y 247.842,Z 530.034,A -85,B 0,C 180,E1 -18806.748,E2 -18806.748} C_VEL
LIN {X 0,Y 248.176,Z 529.146,A -85,B 0,C 180,E1 -18808.377,E2 -18808.377} C_VEL
LIN {X 0,Y 248.344,Z 527.801,A -85,B 0,C 180,E1 -18810,E2 -18810} C_VEL
LIN {X 0,Y 248.483,Z 524.8,A -85,B 0,C 180,E1 -18812.431,E2 -18812.431} C_VEL
LIN {X 0,Y 248.411,Z 520.487,A -85,B 0,C 180,E1 -18814.869,E2 -18814.869} C_VEL
LIN {X 0,Y 248.4,Z 515.776,A -85,B 0,C 180,E1 -18816.932,E2 -18816.932} C_VEL
LIN {X 0,Y 248.407,Z 508.741,A -85,B 0,C 180,E1 -18819.362,E2 -18819.362} C_VEL
LIN {X 0,Y 248.741,Z 501.396,A -85,B 0,C 180,E1 -18821.407,E2 -18821.407} C_VEL
LIN {X 0,Y 249.218,Z 492.228,A -85,B 0,C 180,E1 -18823.453,E2 -18823.453} C_VEL
LIN {X 0,Y 250.006,Z 482.104,A -85,B 0,C 180,E1 -18825.28,E2 -18825.28} C_VEL
LIN {X 0,Y 250.545,Z 471.84,A -85,B 0,C 180,E1 -18826.745,E2 -18826.745} C_VEL
LIN {X 0,Y 249.721,Z 460.328,A -85,B 0,C 180,E1 -18828.034,E2 -18828.034} C_VEL
LIN {X 0,Y 249.068,Z 448.388,A -85,B 0,C 180,E1 -18829.042,E2 -18829.042} C_VEL
LIN {X 0,Y 248.951,Z 437.319,A -85,B 0,C 180,E1 -18829.748,E2 -18829.748} C_VEL
LIN {X 0,Y 251.073,Z 424.515,A -85,B 0,C 180,E1 -18835.713,E2 -18835.713} C_VEL
LIN {X 0,Y 253.61,Z 413.571,A -85,B 0,C 180,E1 -18840.788,E2 -18840.788} C_VEL
LIN {X 0,Y 253.67,Z 411.511,A -85,B 0,C 180,E1 -18841.762,E2 -18841.762} C_VEL
LIN {X 0,Y 251.817,Z 403.045,A -85,B 0,C 180,E1 -18845.966,E2 -18845.966} C_VEL
LIN {X 0,Y 250.078,Z 394.736,A -85,B 0,C 180,E1 -18850.269,E2 -18850.269} C_VEL
LIN {X 0,Y 249.099,Z 389.458,A -85,B 0,C 180,E1 -18853.237,E2 -18853.237} C_VEL
LIN {X 0,Y 249.019,Z 389.461,A -85,B 0,C 180,E1 -18857.363,E2 -18857.363} C_VEL
LIN {X 0,Y 249.039,Z 389.462,A -85,B 0,C 180,E1 -18861.622,E2 -18861.622} C_VEL
LIN {X 0,Y 249.062,Z 389.458,A -85,B 0,C 180,E1 -18865.642,E2 -18865.642} C_VEL
LIN {X 0,Y 249.048,Z 389.461,A -85,B 0,C 180,E1 -18869.473,E2 -18869.473} C_VEL
LIN {X 0,Y 249.072,Z 389.456,A -85,B 0,C 180,E1 -18873.162,E2 -18873.162} C_VEL
LIN {X 0,Y 249.08,Z 389.456,A -85,B 0,C 180,E1 -18876.733,E2 -18876.733} C_VEL
LIN {X 0,Y 249.112,Z 389.453,A -85,B 0,C 180,E1 -18880.212,E2 -18880.212} C_VEL
LIN {X 0,Y 249.242,Z 389.437,A -85,B 0,C 180,E1 -18883.622,E2 -18883.622} C_VEL
LIN {X 0,Y 249.254,Z 389.434,A -85,B 0,C 180,E1 -18888.617,E2 -18888.617} C_VEL
LIN {X 0,Y 249.485,Z 389.407,A -85,B 0,C 180,E1 -18891.903,E2 -18891.903} C_VEL
LIN {X 0,Y 249.442,Z 389.411,A -85,B 0,C 180,E1 -18896.77,E2 -18896.77} C_VEL
LIN {X 0,Y 249.73,Z 389.374,A -85,B 0,C 180,E1 -18900,E2 -18900} C_VEL
LIN {X 0,Y 249.437,Z 389.414,A -85,B 0,C 180,E1 -18903.23,E2 -18903.23} C_VEL
LIN {X 0,Y 249.485,Z 389.404,A -85,B 0,C 180,E1 -18908.097,E2 -18908.097} C_VEL
LIN {X 0,Y 249.254,Z 389.438,A -85,B 0,C 180,E1 -18911.383,E2 -18911.383} C_VEL
LIN {X 0,Y 249.242,Z 389.434,A -85,B 0,C 180,E1 -18916.378,E2 -18916.378} C_VEL
LIN {X 0,Y 249.088,Z 389.457,A -85,B 0,C 180,E1 -18921.518,E2 -18921.518} C_VEL
LIN {X 0,Y 249.131,Z 389.449,A -85,B 0,C 180,E1 -18925.482,E2 -18925.482} C_VEL
LIN {X 0,Y 249.084,Z 389.46,A -85,B 0,C 180,E1 -18928.994,E2 -18928.994} C_VEL
LIN {X 0,Y 249.031,Z 389.463,A -85,B 0,C 180,E1 -18932.426,E2 -18932.426} C_VEL
LIN {X 0,Y 249.049,Z 389.46,A -85,B 0,C 180,E1 -18936.342,E2 -18936.342} C_VEL
LIN {X 0,Y 249.006,Z 389.467,A -85,B 0,C 180,E1 -18940.478,E2 -18940.478} C_VEL
LIN {X 0,Y 249.008,Z 389.468,A -85,B 0,C 180,E1 -18944.878,E2 -18944.878} C_VEL
LIN {X 0,Y 249.019,Z 389.464,A -85,B 0,C 180,E1 -18947.364,E2 -18947.364} C_VEL
LIN {X 0,Y 249.039,Z 389.459,A -85,B 0,C 180,E1 -18951.622,E2 -18951.622} C_VEL
LIN {X 0,Y 249.062,Z 389.458,A -85,B 0,C 180,E1 -18955.643,E2 -18955.643} C_VEL
LIN {X 0,Y 249.052,Z 389.458,A -85,B 0,C 180,E1 -18959.473,E2 -18959.473} C_VEL
LIN {X 0,Y 249.074,Z 389.457,A -85,B 0,C 180,E1 -18963.163,E2 -18963.163} C_VEL
LIN {X 0,Y 249.087,Z 389.456,A -85,B 0,C 180,E1 -18966.734,E2 -18966.734} C_VEL
LIN {X 0,Y 249.133,Z 389.451,A -85,B 0,C 180,E1 -18970.214,E2 -18970.214} C_VEL
LIN {X 0,Y 249.244,Z 389.436,A -85,B 0,C 180,E1 -18973.622,E2 -18973.622} C_VEL
LIN {X 0,Y 249.255,Z 389.435,A -85,B 0,C 180,E1 -18978.617,E2 -18978.617} C_VEL
LIN {X 0,Y 249.482,Z 389.409,A -85,B 0,C 180,E1 -18981.903,E2 -18981.903} C_VEL
LIN {X 0,Y 249.438,Z 389.411,A -85,B 0,C 180,E1 -18986.77,E2 -18986.77} C_VEL
LIN {X 0,Y 249.738,Z 389.379,A -85,B 0,C 180,E1 -18990,E2 -18990} C_VEL
LIN {X 0,Y 249.438,Z 389.411,A -85,B 0,C 180,E1 -18993.231,E2 -18993.231} C_VEL
LIN {X 0,Y 249.456,Z 389.41,A -85,B 0,C 180,E1 -18996.471,E2 -18996.471} C_VEL
LIN {X 0,Y 249.346,Z 389.427,A -85,B 0,C 180,E1 -18999.737,E2 -18999.737} C_VEL
LIN {X 0,Y 249.208,Z 389.439,A -85,B 0,C 180,E1 -19004.704,E2 -19004.704} C_VEL
LIN {X 0,Y 249.142,Z 389.45,A -85,B 0,C 180,E1 -19008.077,E2 -19008.077} C_VEL
LIN {X 0,Y 249.091,Z 389.456,A -85,B 0,C 180,E1 -19011.518,E2 -19011.518} C_VEL
LIN {X 0,Y 249.133,Z 389.453,A -85,B 0,C 180,E1 -19015.482,E2 -19015.482} C_VEL
LIN {X 0,Y 249.082,Z 389.456,A -85,B 0,C 180,E1 -19018.992,E2 -19018.992} C_VEL
LIN {X 0,Y 249.039,Z 389.461,A -85,B 0,C 180,E1 -19022.425,E2 -19022.425} C_VEL
LIN {X 0,Y 249.072,Z 389.457,A -85,B 0,C 180,E1 -19026.339,E2 -19026.339} C_VEL
LIN {X 0,Y 249.028,Z 389.462,A -85,B 0,C 180,E1 -19030.474,E2 -19030.474} C_VEL
LIN {X 0,Y 249.01,Z 389.467,A -85,B 0,C 180,E1 -19034.878,E2 -19034.878} C_VEL
LIN {X 0,Y 249.021,Z 389.465,A -85,B 0,C 180,E1 -19037.364,E2 -19037.364} C_VEL
LIN {X 0,Y 249.049,Z 389.46,A -85,B 0,C 180,E1 -19042.199,E2 -19042.199} C_VEL
LIN {X 0,Y 249.13,Z 389.448,A -85,B 0,C 180,E1 -19045.653,E2 -19045.653} C_VEL
LIN {X 0,Y 249.338,Z 389.522,A -85,B 0,C 180,E1 -19047.902,E2 -19047.902} C_VEL
LIN {X 0,Y 249.452,Z 391.6,A -85,B 0,C 180,E1 -19049.527,E2 -19049.527} C_VEL
LIN {X 0,Y 249.016,Z 396.41,A -85,B 0,C 180,E1 -19053.155,E2 -19053.155} C_VEL
LIN {X 0,Y 248.472,Z 402.354,A -85,B 0,C 180,E1 -19057.552,E2 -19057.552} C_VEL
LIN {X 0,Y 248.079,Z 408.307,A -85,B 0,C 180,E1 -19061.843,E2 -19061.843} C_VEL
LIN {X 0,Y 247.771,Z 414.258,A -85,B 0,C 180,E1 -19066.048,E2 -19066.048} C_VEL
LIN {X 0,Y 247.745,Z 415.791,A -85,B 0,C 180,E1 -19067.039,E2 -19067.039} C_VEL
LIN {X 0,Y 248.816,Z 428.203,A -85,B 0,C 180,E1 -19068.183,E2 -19068.183} C_VEL
LIN {X 0,Y 249.439,Z 433.85,A -85,B 0,C 180,E1 -19068.831,E2 -19068.831} C_VEL
LIN {X 0,Y 248.968,Z 444.161,A -85,B 0,C 180,E1 -19070.249,E2 -19070.249} C_VEL
LIN {X 0,Y 248.521,Z 453.6,A -85,B 0,C 180,E1 -19071.871,E2 -19071.871} C_VEL
LIN {X 0,Y 248.246,Z 463.074,A -85,B 0,C 180,E1 -19073.906,E2 -19073.906} C_VEL
LIN {X 0,Y 247.776,Z 470.553,A -85,B 0,C 180,E1 -19075.934,E2 -19075.934} C_VEL
LIN {X 0,Y 247.541,Z 477.523,A -85,B 0,C 180,E1 -19078.373,E2 -19078.373} C_VEL
LIN {X 0,Y 247.769,Z 482.786,A -85,B 0,C 180,E1 -19080.813,E2 -19080.813} C_VEL
LIN {X 0,Y 248.296,Z 486.537,A -85,B 0,C 180,E1 -19083.245,E2 -19083.245} C_VEL
LIN {X 0,Y 248.885,Z 488.255,A -85,B 0,C 180,E1 -19084.86,E2 -19084.86} C_VEL
LIN {X 0,Y 249.722,Z 489.401,A -85,B 0,C 180,E1 -19086.464,E2 -19086.464} C_VEL
LIN {X 0,Y 250.745,Z 489.971,A -85,B 0,C 180,E1 -19088.056,E2 -19088.056} C_VEL
LIN {X 0,Y 252.01,Z 489.935,A -85,B 0,C 180,E1 -19089.632,E2 -19089.632} C_VEL
LIN {X 0,Y 253.561,Z 489.342,A -85,B 0,C 180,E1 -19091.188,E2 -19091.188} C_VEL
LIN {X 0,Y 255.232,Z 488.224,A -85,B 0,C 180,E1 -19092.726,E2 -19092.726} C_VEL
LIN {X 0,Y 258.044,Z 485.442,A -85,B 0,C 180,E1 -19094.995,E2 -19094.995} C_VEL
LIN {X 0,Y 261.31,Z 481.334,A -85,B 0,C 180,E1 -19097.208,E2 -19097.208} C_VEL
LIN {X 0,Y 264.93,Z 475.805,A -85,B 0,C 180,E1 -19099.366,E2 -19099.366} C_VEL
LIN {X 0,Y 268.142,Z 469.976,A -85,B 0,C 180,E1 -19101.124,E2 -19101.124} C_VEL
LIN {X 0,Y 268.919,Z 463.349,A -85,B 0,C 180,E1 -19103.528,E2 -19103.528} C_VEL
LIN {X 0,Y 268.859,Z 456.787,A -85,B 0,C 180,E1 -19105.944,E2 -19105.944} C_VEL
LIN {X 0,Y 268.058,Z 449.816,A -85,B 0,C 180,E1 -19108.693,E2 -19108.693} C_VEL
LIN {X 0,Y 267.169,Z 445.16,A -85,B 0,C 180,E1 -19110.799,E2 -19110.799} C_VEL
LIN {X 0,Y 266.367,Z 442.135,A -85,B 0,C 180,E1 -19112.401,E2 -19112.401} C_VEL
LIN {X 0,Y 265.154,Z 438.761,A -85,B 0,C 180,E1 -19114.747,E2 -19114.747} C_VEL
LIN {X 0,Y 263.73,Z 436.465,A -85,B 0,C 180,E1 -19117.801,E2 -19117.801} C_VEL
LIN {X 0,Y 263.35,Z 435.403,A -85,B 0,C 180,E1 -19119.828,E2 -19119.828} C_VEL
LIN {X 0,Y 263.272,Z 435.156,A -85,B 0,C 180,E1 -19121.865,E2 -19121.865} C_VEL
LIN {X 0,Y 263.324,Z 435.448,A -85,B 0,C 180,E1 -19122.753,E2 -19122.753} C_VEL
LIN {X 0,Y 263.233,Z 436.651,A -85,B 0,C 180,E1 -19124.008,E2 -19124.008} C_VEL
LIN {X 0,Y 262.892,Z 438.963,A -85,B 0,C 180,E1 -19125.2,E2 -19125.2} C_VEL
LIN {X 0,Y 262.247,Z 444.753,A -85,B 0,C 180,E1 -19127.507,E2 -19127.507} C_VEL
LIN {X 0,Y 262.465,Z 447.204,A -85,B 0,C 180,E1 -19128.706,E2 -19128.706} C_VEL
LIN {X 0,Y 262.718,Z 447.82,A -85,B 0,C 180,E1 -19129.118,E2 -19129.118} C_VEL
LIN {X 0,Y 263.883,Z 449.775,A -85,B 0,C 180,E1 -19130.566,E2 -19130.566} C_VEL
LIN {X 0,Y 266.396,Z 456.206,A -85,B 0,C 180,E1 -19133.621,E2 -19133.621} C_VEL
LIN {X 0,Y 266.734,Z 457.67,A -85,B 0,C 180,E1 -19134.125,E2 -19134.125} C_VEL
LIN {X 0,Y 266.153,Z 467.645,A -85,B 0,C 180,E1 -19136.477,E2 -19136.477} C_VEL
LIN {X 0,Y 264.64,Z 478.086,A -85,B 0,C 180,E1 -19138.819,E2 -19138.819} C_VEL
LIN {X 0,Y 262.934,Z 485.086,A -85,B 0,C 180,E1 -19140.364,E2 -19140.364} C_VEL
LIN {X 0,Y 259.754,Z 493.23,A -85,B 0,C 180,E1 -19142.178,E2 -19142.178} C_VEL
LIN {X 0,Y 255.331,Z 501.859,A -85,B 0,C 180,E1 -19144.308,E2 -19144.308} C_VEL
LIN {X 0,Y 252.062,Z 507.835,A -85,B 0,C 180,E1 -19146.153,E2 -19146.153} C_VEL
LIN {X 0,Y 247.629,Z 515.625,A -85,B 0,C 180,E1 -19149.221,E2 -19149.221} C_VEL
LIN {X 0,Y 245.038,Z 520.2,A -85,B 0,C 180,E1 -19151.609,E2 -19151.609} C_VEL
LIN {X 0,Y 242.536,Z 524.798,A -85,B 0,C 180,E1 -19154.882,E2 -19154.882} C_VEL
LIN {X 0,Y 241.518,Z 526.53,A -85,B 0,C 180,E1 -19156.538,E2 -19156.538} C_VEL
LIN {X 0,Y 240.512,Z 528.823,A -85,B 0,C 180,E1 -19159.902,E2 -19159.902} C_VEL
LIN {X 0,Y 240.388,Z 529.65,A -85,B 0,C 180,E1 -19163.284,E2 -19163.284} C_VEL
LIN {X 0,Y 240.81,Z 528.884,A -85,B 0,C 180,E1 -19166.653,E2 -19166.653} C_VEL
LIN {X 0,Y 241.174,Z 527.9,A -85,B 0,C 180,E1 -19168.33,E2 -19168.33} C_VEL
LIN {X 0,Y 241.385,Z 526.395,A -85,B 0,C 180,E1 -19170,E2 -19170} C_VEL
LIN {X 0,Y 241.541,Z 523.176,A -85,B 0,C 180,E1 -19172.501,E2 -19172.501} C_VEL
LIN {X 0,Y 241.448,Z 518.645,A -85,B 0,C 180,E1 -19175.009,E2 -19175.009} C_VEL
LIN {X 0,Y 241.401,Z 512.608,A -85,B 0,C 180,E1 -19177.54,E2 -19177.54} C_VEL
LIN {X 0,Y 241.541,Z 504.891,A -85,B 0,C 180,E1 -19180.054,E2 -19180.054} C_VEL
LIN {X 0,Y 241.96,Z 496.833,A -85,B 0,C 180,E1 -19182.156,E2 -19182.156} C_VEL
LIN {X 0,Y 242.49,Z 486.745,A -85,B 0,C 180,E1 -19184.261,E2 -19184.261} C_VEL
LIN {X 0,Y 243.276,Z 476.789,A -85,B 0,C 180,E1 -19185.929,E2 -19185.929} C_VEL
LIN {X 0,Y 243.387,Z 470.617,A -85,B 0,C 180,E1 -19186.783,E2 -19186.783} C_VEL
LIN {X 0,Y 242.564,Z 459.129,A -85,B 0,C 180,E1 -19188.088,E2 -19188.088} C_VEL
LIN {X 0,Y 241.891,Z 446.203,A -85,B 0,C 180,E1 -19189.188,E2 -19189.188} C_VEL
LIN {X 0,Y 241.888,Z 437.002,A -85,B 0,C 180,E1 -19189.796,E2 -19189.796} C_VEL
LIN {X 0,Y 243.912,Z 425.009,A -85,B 0,C 180,E1 -19195.607,E2 -19195.607} C_VEL
LIN {X 0,Y 246.517,Z 414.049,A -85,B 0,C 180,E1 -19200.875,E2 -19200.875} C_VEL
LIN {X 0,Y 246.515,Z 411.852,A -85,B 0,C 180,E1 -19201.957,E2 -19201.957} C_VEL
LIN {X 0,Y 244.313,Z 401.713,A -85,B 0,C 180,E1 -19207.163,E2 -19207.163} C_VEL
LIN {X 0,Y 242.389,Z 392.275,A -85,B 0,C 180,E1 -19212.323,E2 -19212.323} C_VEL
LIN {X 0,Y 242.047,Z 390.337,A -85,B 0,C 180,E1 -19213.457,E2 -19213.457} C_VEL
LIN {X 0,Y 241.945,Z 390.346,A -85,B 0,C 180,E1 -19218.079,E2 -19218.079} C_VEL
LIN {X 0,Y 242.002,Z 390.34,A -85,B 0,C 180,E1 -19222.42,E2 -19222.42} C_VEL
LIN {X 0,Y 241.992,Z 390.339,A -85,B 0,C 180,E1 -19226.509,E2 -19226.509} C_VEL
LIN {X 0,Y 242.014,Z 390.337,A -85,B 0,C 180,E1 -19230.597,E2 -19230.597} C_VEL
LIN {X 0,Y 242.068,Z 390.33,A -85,B 0,C 180,E1 -19234.183,E2 -19234.183} C_VEL
LIN {X 0,Y 242.054,Z 390.333,A -85,B 0,C 180,E1 -19238.297,E2 -19238.297} C_VEL
LIN {X 0,Y 242.164,Z 390.316,A -85,B 0,C 180,E1 -19243.278,E2 -19243.278} C_VEL
LIN {X 0,Y 242.187,Z 390.315,A -85,B 0,C 180,E1 -19248.28,E2 -19248.28} C_VEL
LIN {X 0,Y 242.436,Z 390.285,A -85,B 0,C 180,E1 -19251.666,E2 -19251.666} C_VEL
LIN {X 0,Y 242.263,Z 390.306,A -85,B 0,C 180,E1 -19255.007,E2 -19255.007} C_VEL
LIN {X 0,Y 242.64,Z 390.257,A -85,B 0,C 180,E1 -19258.34,E2 -19258.34} C_VEL
LIN {X 0,Y 242.637,Z 390.261,A -85,B 0,C 180,E1 -19261.66,E2 -19261.66} C_VEL
LIN {X 0,Y 242.43,Z 390.284,A -85,B 0,C 180,E1 -19266.743,E2 -19266.743} C_VEL
LIN {X 0,Y 242.346,Z 390.295,A -85,B 0,C 180,E1 -19270.02,E2 -19270.02} C_VEL
LIN {X 0,Y 242.168,Z 390.321,A -85,B 0,C 180,E1 -19275.141,E2 -19275.141} C_VEL
LIN {X 0,Y 242.074,Z 390.328,A -85,B 0,C 180,E1 -19278.624,E2 -19278.624} C_VEL
LIN {X 0,Y 242.014,Z 390.337,A -85,B 0,C 180,E1 -19282.18,E2 -19282.18} C_VEL
LIN {X 0,Y 242.067,Z 390.328,A -85,B 0,C 180,E1 -19285.838,E2 -19285.838} C_VEL
LIN {X 0,Y 242.031,Z 390.335,A -85,B 0,C 180,E1 -19289.58,E2 -19289.58} C_VEL
LIN {X 0,Y 241.981,Z 390.339,A -85,B 0,C 180,E1 -19293.493,E2 -19293.493} C_VEL
LIN {X 0,Y 241.99,Z 390.34,A -85,B 0,C 180,E1 -19297.582,E2 -19297.582} C_VEL
LIN {X 0,Y 241.939,Z 390.344,A -85,B 0,C 180,E1 -19301.922,E2 -19301.922} C_VEL
LIN {X 0,Y 241.937,Z 390.349,A -85,B 0,C 180,E1 -19306.571,E2 -19306.571} C_VEL
LIN {X 0,Y 241.973,Z 390.342,A -85,B 0,C 180,E1 -19310.285,E2 -19310.285} C_VEL
LIN {X 0,Y 242.038,Z 390.337,A -85,B 0,C 180,E1 -19314.498,E2 -19314.498} C_VEL
LIN {X 0,Y 241.977,Z 390.344,A -85,B 0,C 180,E1 -19318.481,E2 -19318.481} C_VEL
LIN {X 0,Y 242.008,Z 390.339,A -85,B 0,C 180,E1 -19322.313,E2 -19322.313} C_VEL
LIN {X 0,Y 242.062,Z 390.332,A -85,B 0,C 180,E1 -19326.017,E2 -19326.017} C_VEL
LIN {X 0,Y 242.063,Z 390.329,A -85,B 0,C 180,E1 -19329.611,E2 -19329.611} C_VEL
LIN {X 0,Y 242.165,Z 390.318,A -85,B 0,C 180,E1 -19333.278,E2 -19333.278} C_VEL
LIN {X 0,Y 242.189,Z 390.317,A -85,B 0,C 180,E1 -19338.28,E2 -19338.28} C_VEL
LIN {X 0,Y 242.429,Z 390.286,A -85,B 0,C 180,E1 -19341.666,E2 -19341.666} C_VEL
LIN {X 0,Y 242.261,Z 390.304,A -85,B 0,C 180,E1 -19345.008,E2 -19345.008} C_VEL
LIN {X 0,Y 242.639,Z 390.261,A -85,B 0,C 180,E1 -19348.341,E2 -19348.341} C_VEL
LIN {X 0,Y 242.639,Z 390.261,A -85,B 0,C 180,E1 -19351.66,E2 -19351.66} C_VEL
LIN {X 0,Y 242.426,Z 390.285,A -85,B 0,C 180,E1 -19356.659,E2 -19356.659} C_VEL
LIN {X 0,Y 242.27,Z 390.307,A -85,B 0,C 180,E1 -19360.024,E2 -19360.024} C_VEL
LIN {X 0,Y 242.17,Z 390.317,A -85,B 0,C 180,E1 -19365.141,E2 -19365.141} C_VEL
LIN {X 0,Y 242.077,Z 390.328,A -85,B 0,C 180,E1 -19368.624,E2 -19368.624} C_VEL
LIN {X 0,Y 242.017,Z 390.336,A -85,B 0,C 180,E1 -19372.18,E2 -19372.18} C_VEL
LIN {X 0,Y 242.069,Z 390.332,A -85,B 0,C 180,E1 -19375.838,E2 -19375.838} C_VEL
LIN {X 0,Y 242.031,Z 390.335,A -85,B 0,C 180,E1 -19379.58,E2 -19379.58} C_VEL
LIN {X 0,Y 241.994,Z 390.343,A -85,B 0,C 180,E1 -19383.491,E2 -19383.491} C_VEL
LIN {X 0,Y 242.005,Z 390.338,A -85,B 0,C 180,E1 -19387.579,E2 -19387.579} C_VEL
LIN {X 0,Y 241.947,Z 390.346,A -85,B 0,C 180,E1 -19391.921,E2 -19391.921} C_VEL
LIN {X 0,Y 241.939,Z 390.344,A -85,B 0,C 180,E1 -19396.571,E2 -19396.571} C_VEL
LIN {X 0,Y 241.959,Z 390.343,A -85,B 0,C 180,E1 -19400.281,E2 -19400.281} C_VEL
LIN {X 0,Y 242.039,Z 390.333,A -85,B 0,C 180,E1 -19404.498,E2 -19404.498} C_VEL
LIN {X 0,Y 242.281,Z 390.437,A -85,B 0,C 180,E1 -19407.921,E2 -19407.921} C_VEL
LIN {X 0,Y 242.401,Z 392.451,A -85,B 0,C 180,E1 -19409.51,E2 -19409.51} C_VEL
LIN {X 0,Y 241.939,Z 397.277,A -85,B 0,C 180,E1 -19413.24,E2 -19413.24} C_VEL
LIN {X 0,Y 241.37,Z 403.264,A -85,B 0,C 180,E1 -19417.758,E2 -19417.758} C_VEL
LIN {X 0,Y 240.965,Z 409.244,A -85,B 0,C 180,E1 -19422.167,E2 -19422.167} C_VEL
LIN {X 0,Y 240.663,Z 415.978,A -85,B 0,C 180,E1 -19427.027,E2 -19427.027} C_VEL
LIN {X 0,Y 241.775,Z 428.886,A -85,B 0,C 180,E1 -19428.259,E2 -19428.259} C_VEL
LIN {X 0,Y 242.332,Z 434.477,A -85,B 0,C 180,E1 -19428.923,E2 -19428.923} C_VEL
LIN {X 0,Y 241.796,Z 446.087,A -85,B 0,C 180,E1 -19430.59,E2 -19430.59} C_VEL
LIN {X 0,Y 241.263,Z 456.386,A -85,B 0,C 180,E1 -19432.489,E2 -19432.489} C_VEL
LIN {X 0,Y 241.126,Z 463.632,A -85,B 0,C 180,E1 -19434.145,E2 -19434.145} C_VEL
LIN {X 0,Y 240.64,Z 471.054,A -85,B 0,C 180,E1 -19436.232,E2 -19436.232} C_VEL
LIN {X 0,Y 240.46,Z 478.111,A -85,B 0,C 180,E1 -19438.744,E2 -19438.744} C_VEL
LIN {X 0,Y 240.667,Z 482.655,A -85,B 0,C 180,E1 -19440.837,E2 -19440.837} C_VEL
LIN {X 0,Y 241.21,Z 486.698,A -85,B 0,C 180,E1 -19443.341,E2 -19443.341} C_VEL
LIN {X 0,Y 241.85,Z 488.629,A -85,B 0,C 180,E1 -19445.001,E2 -19445.001} C_VEL
LIN {X 0,Y 242.699,Z 489.961,A -85,B 0,C 180,E1 -19446.652,E2 -19446.652} C_VEL
LIN {X 0,Y 243.773,Z 490.728,A -85,B 0,C 180,E1 -19448.288,E2 -19448.288} C_VEL
LIN {X 0,Y 245.082,Z 490.942,A -85,B 0,C 180,E1 -19449.907,E2 -19449.907} C_VEL
LIN {X 0,Y 246.708,Z 490.556,A -85,B 0,C 180,E1 -19451.502,E2 -19451.502} C_VEL
LIN {X 0,Y 248.437,Z 489.634,A -85,B 0,C 180,E1 -19453.08,E2 -19453.08} C_VEL
LIN {X 0,Y 251.406,Z 487.25,A -85,B 0,C 180,E1 -19455.401,E2 -19455.401} C_VEL
LIN {X 0,Y 254.803,Z 483.547,A -85,B 0,C 180,E1 -19457.662,E2 -19457.662} C_VEL
LIN {X 0,Y 259.253,Z 477.499,A -85,B 0,C 180,E1 -19460.221,E2 -19460.221} C_VEL
LIN {X 0,Y 262.094,Z 473.089,A -85,B 0,C 180,E1 -19461.636,E2 -19461.636} C_VEL
LIN {X 0,Y 263.196,Z 468.003,A -85,B 0,C 180,E1 -19463.612,E2 -19463.612} C_VEL
LIN {X 0,Y 263.582,Z 462.378,A -85,B 0,C 180,E1 -19465.877,E2 -19465.877} C_VEL
LIN {X 0,Y 263.505,Z 456.495,A -85,B 0,C 180,E1 -19468.339,E2 -19468.339} C_VEL
LIN {X 0,Y 262.874,Z 450.532,A -85,B 0,C 180,E1 -19471.181,E2 -19471.181} C_VEL
LIN {X 0,Y 262.517,Z 448.422,A -85,B 0,C 180,E1 -19472.373,E2 -19472.373} C_VEL
LIN {X 0,Y 261.757,Z 445.674,A -85,B 0,C 180,E1 -19474.322,E2 -19474.322} C_VEL
LIN {X 0,Y 260.971,Z 443.778,A -85,B 0,C 180,E1 -19476.332,E2 -19476.332} C_VEL
LIN {X 0,Y 260.422,Z 442.451,A -85,B 0,C 180,E1 -19478.498,E2 -19478.498} C_VEL
LIN {X 0,Y 260.271,Z 441.661,A -85,B 0,C 180,E1 -19480.88,E2 -19480.88} C_VEL
LIN {X 0,Y 260.445,Z 442.068,A -85,B 0,C 180,E1 -19483.232,E2 -19483.232} C_VEL
LIN {X 0,Y 261.006,Z 443.578,A -85,B 0,C 180,E1 -19485.565,E2 -19485.565} C_VEL
LIN {X 0,Y 262.718,Z 447.82,A -85,B 0,C 180,E1 -19489.118,E2 -19489.118} C_VEL
LIN {X 0,Y 263.327,Z 450.113,A -85,B 0,C 180,E1 -19490.3,E2 -19490.3} C_VEL
LIN {X 0,Y 263.396,Z 453.39,A -85,B 0,C 180,E1 -19491.384,E2 -19491.384} C_VEL
LIN {X 0,Y 263.2,Z 455.908,A -85,B 0,C 180,E1 -19492.056,E2 -19492.056} C_VEL
LIN {X 0,Y 261.637,Z 466.966,A -85,B 0,C 180,E1 -19494.683,E2 -19494.683} C_VEL
LIN {X 0,Y 260.217,Z 475.838,A -85,B 0,C 180,E1 -19496.852,E2 -19496.852} C_VEL
LIN {X 0,Y 258.202,Z 484.14,A -85,B 0,C 180,E1 -19498.858,E2 -19498.858} C_VEL
LIN {X 0,Y 255.822,Z 490.596,A -85,B 0,C 180,E1 -19500.363,E2 -19500.363} C_VEL
LIN {X 0,Y 252.076,Z 497.937,A -85,B 0,C 180,E1 -19502.16,E2 -19502.16} C_VEL
LIN {X 0,Y 246.843,Z 506.619,A -85,B 0,C 180,E1 -19504.718,E2 -19504.718} C_VEL
LIN {X 0,Y 243.267,Z 512.627,A -85,B 0,C 180,E1 -19507.044,E2 -19507.044} C_VEL
LIN {X 0,Y 239.502,Z 518.357,A -85,B 0,C 180,E1 -19509.887,E2 -19509.887} C_VEL
LIN {X 0,Y 236.825,Z 522.646,A -85,B 0,C 180,E1 -19512.737,E2 -19512.737} C_VEL
LIN {X 0,Y 234.601,Z 526.112,A -85,B 0,C 180,E1 -19516.133,E2 -19516.133} C_VEL
LIN {X 0,Y 233.507,Z 528.149,A -85,B 0,C 180,E1 -19519.596,E2 -19519.596} C_VEL
LIN {X 0,Y 233.35,Z 528.674,A -85,B 0,C 180,E1 -19523.08,E2 -19523.08} C_VEL
LIN {X 0,Y 233.492,Z 528.386,A -85,B 0,C 180,E1 -19524.819,E2 -19524.819} C_VEL
LIN {X 0,Y 233.791,Z 527.669,A -85,B 0,C 180,E1 -19526.553,E2 -19526.553} C_VEL
LIN {X 0,Y 234.211,Z 526.545,A -85,B 0,C 180,E1 -19528.28,E2 -19528.28} C_VEL
LIN {X 0,Y 234.489,Z 523.909,A -85,B 0,C 180,E1 -19530.858,E2 -19530.858} C_VEL
LIN {X 0,Y 234.573,Z 520.049,A -85,B 0,C 180,E1 -19533.435,E2 -19533.435} C_VEL
LIN {X 0,Y 234.522,Z 514.796,A -85,B 0,C 180,E1 -19536.02,E2 -19536.02} C_VEL
LIN {X 0,Y 234.447,Z 507.847,A -85,B 0,C 180,E1 -19538.62,E2 -19538.62} C_VEL
LIN {X 0,Y 234.704,Z 500.674,A -85,B 0,C 180,E1 -19540.786,E2 -19540.786} C_VEL
LIN {X 0,Y 235.128,Z 491.764,A -85,B 0,C 180,E1 -19542.954,E2 -19542.954} C_VEL
LIN {X 0,Y 235.809,Z 481.908,A -85,B 0,C 180,E1 -19544.895,E2 -19544.895} C_VEL
LIN {X 0,Y 236.425,Z 472.389,A -85,B 0,C 180,E1 -19546.403,E2 -19546.403} C_VEL
LIN {X 0,Y 235.558,Z 460.251,A -85,B 0,C 180,E1 -19547.885,E2 -19547.885} C_VEL
LIN {X 0,Y 234.867,Z 448.335,A -85,B 0,C 180,E1 -19548.99,E2 -19548.99} C_VEL
LIN {X 0,Y 234.8,Z 436.752,A -85,B 0,C 180,E1 -19549.792,E2 -19549.792} C_VEL
LIN {X 0,Y 236.725,Z 425.445,A -85,B 0,C 180,E1 -19555.498,E2 -19555.498} C_VEL
LIN {X 0,Y 239.341,Z 414.759,A -85,B 0,C 180,E1 -19560.816,E2 -19560.816} C_VEL
LIN {X 0,Y 239.475,Z 412.634,A -85,B 0,C 180,E1 -19561.887,E2 -19561.887} C_VEL
LIN {X 0,Y 237.398,Z 403.209,A -85,B 0,C 180,E1 -19566.935,E2 -19566.935} C_VEL
LIN {X 0,Y 235.595,Z 394.509,A -85,B 0,C 180,E1 -19571.775,E2 -19571.775} C_VEL
LIN {X 0,Y 234.982,Z 391.218,A -85,B 0,C 180,E1 -19573.773,E2 -19573.773} C_VEL
LIN {X 0,Y 234.898,Z 391.223,A -85,B 0,C 180,E1 -19578.835,E2 -19578.835} C_VEL
LIN {X 0,Y 234.955,Z 391.216,A -85,B 0,C 180,E1 -19581.086,E2 -19581.086} C_VEL
LIN {X 0,Y 234.961,Z 391.213,A -85,B 0,C 180,E1 -19585.367,E2 -19585.367} C_VEL
LIN {X 0,Y 234.923,Z 391.22,A -85,B 0,C 180,E1 -19589.431,E2 -19589.431} C_VEL
LIN {X 0,Y 234.994,Z 391.212,A -85,B 0,C 180,E1 -19593.794,E2 -19593.794} C_VEL
LIN {X 0,Y 235.012,Z 391.209,A -85,B 0,C 180,E1 -19598.97,E2 -19598.97} C_VEL
LIN {X 0,Y 235.097,Z 391.195,A -85,B 0,C 180,E1 -19603.059,E2 -19603.059} C_VEL
LIN {X 0,Y 235.147,Z 391.194,A -85,B 0,C 180,E1 -19607.924,E2 -19607.924} C_VEL
LIN {X 0,Y 235.391,Z 391.162,A -85,B 0,C 180,E1 -19611.415,E2 -19611.415} C_VEL
LIN {X 0,Y 235.407,Z 391.159,A -85,B 0,C 180,E1 -19613.141,E2 -19613.141} C_VEL
LIN {X 0,Y 235.6,Z 391.134,A -85,B 0,C 180,E1 -19618.291,E2 -19618.291} C_VEL
LIN {X 0,Y 235.597,Z 391.138,A -85,B 0,C 180,E1 -19621.709,E2 -19621.709} C_VEL
LIN {X 0,Y 235.407,Z 391.16,A -85,B 0,C 180,E1 -19626.859,E2 -19626.859} C_VEL
LIN {X 0,Y 235.254,Z 391.178,A -85,B 0,C 180,E1 -19630.326,E2 -19630.326} C_VEL
LIN {X 0,Y 235.115,Z 391.196,A -85,B 0,C 180,E1 -19635.606,E2 -19635.606} C_VEL
LIN {X 0,Y 235.01,Z 391.212,A -85,B 0,C 180,E1 -19639.206,E2 -19639.206} C_VEL
LIN {X 0,Y 234.962,Z 391.217,A -85,B 0,C 180,E1 -19642.883,E2 -19642.883} C_VEL
LIN {X 0,Y 234.97,Z 391.213,A -85,B 0,C 180,E1 -19646.657,E2 -19646.657} C_VEL
LIN {X 0,Y 234.932,Z 391.22,A -85,B 0,C 180,E1 -19650.568,E2 -19650.568} C_VEL
LIN {X 0,Y 234.931,Z 391.218,A -85,B 0,C 180,E1 -19654.638,E2 -19654.638} C_VEL
LIN {X 0,Y 234.942,Z 391.221,A -85,B 0,C 180,E1 -19658.945,E2 -19658.945} C_VEL
LIN {X 0,Y 234.89,Z 391.222,A -85,B 0,C 180,E1 -19663.485,E2 -19663.485} C_VEL
LIN {X 0,Y 234.89,Z 391.226,A -85,B 0,C 180,E1 -19666.515,E2 -19666.515} C_VEL
LIN {X 0,Y 234.956,Z 391.214,A -85,B 0,C 180,E1 -19671.086,E2 -19671.086} C_VEL
LIN {X 0,Y 234.961,Z 391.215,A -85,B 0,C 180,E1 -19675.368,E2 -19675.368} C_VEL
LIN {X 0,Y 234.97,Z 391.213,A -85,B 0,C 180,E1 -19680.158,E2 -19680.158} C_VEL
LIN {X 0,Y 234.995,Z 391.211,A -85,B 0,C 180,E1 -19683.794,E2 -19683.794} C_VEL
LIN {X 0,Y 235.03,Z 391.205,A -85,B 0,C 180,E1 -19688.972,E2 -19688.972} C_VEL
LIN {X 0,Y 235.098,Z 391.198,A -85,B 0,C 180,E1 -19693.059,E2 -19693.059} C_VEL
LIN {X 0,Y 235.15,Z 391.191,A -85,B 0,C 180,E1 -19697.924,E2 -19697.924} C_VEL
LIN {X 0,Y 235.378,Z 391.164,A -85,B 0,C 180,E1 -19701.414,E2 -19701.414} C_VEL
LIN {X 0,Y 235.405,Z 391.159,A -85,B 0,C 180,E1 -19703.142,E2 -19703.142} C_VEL
LIN {X 0,Y 235.599,Z 391.138,A -85,B 0,C 180,E1 -19708.291,E2 -19708.291} C_VEL
LIN {X 0,Y 235.598,Z 391.138,A -85,B 0,C 180,E1 -19711.71,E2 -19711.71} C_VEL
LIN {X 0,Y 235.376,Z 391.163,A -85,B 0,C 180,E1 -19716.86,E2 -19716.86} C_VEL
LIN {X 0,Y 235.217,Z 391.183,A -85,B 0,C 180,E1 -19720.328,E2 -19720.328} C_VEL
LIN {X 0,Y 235.117,Z 391.198,A -85,B 0,C 180,E1 -19725.607,E2 -19725.607} C_VEL
LIN {X 0,Y 235.012,Z 391.21,A -85,B 0,C 180,E1 -19729.206,E2 -19729.206} C_VEL
LIN {X 0,Y 234.965,Z 391.213,A -85,B 0,C 180,E1 -19732.883,E2 -19732.883} C_VEL
LIN {X 0,Y 234.972,Z 391.214,A -85,B 0,C 180,E1 -19736.658,E2 -19736.658} C_VEL
LIN {X 0,Y 234.934,Z 391.216,A -85,B 0,C 180,E1 -19740.568,E2 -19740.568} C_VEL
LIN {X 0,Y 234.963,Z 391.215,A -85,B 0,C 180,E1 -19744.633,E2 -19744.633} C_VEL
LIN {X 0,Y 234.944,Z 391.216,A -85,B 0,C 180,E1 -19748.945,E2 -19748.945} C_VEL
LIN {X 0,Y 234.892,Z 391.226,A -85,B 0,C 180,E1 -19753.485,E2 -19753.485} C_VEL
LIN {X 0,Y 234.892,Z 391.222,A -85,B 0,C 180,E1 -19756.515,E2 -19756.515} C_VEL
LIN {X 0,Y 234.922,Z 391.223,A -85,B 0,C 180,E1 -19761.079,E2 -19761.079} C_VEL
LIN {X 0,Y 235.013,Z 391.207,A -85,B 0,C 180,E1 -19765.376,E2 -19765.376} C_VEL
LIN {X 0,Y 235.256,Z 391.374,A -85,B 0,C 180,E1 -19767.977,E2 -19767.977} C_VEL
LIN {X 0,Y 235.273,Z 393.921,A -85,B 0,C 180,E1 -19770.03,E2 -19770.03} C_VEL
LIN {X 0,Y 234.74,Z 398.881,A -85,B 0,C 180,E1 -19773.921,E2 -19773.921} C_VEL
LIN {X 0,Y 234.211,Z 405.37,A -85,B 0,C 180,E1 -19778.894,E2 -19778.894} C_VEL
LIN {X 0,Y 233.777,Z 411.513,A -85,B 0,C 180,E1 -19783.495,E2 -19783.495} C_VEL
LIN {X 0,Y 233.569,Z 416.298,A -85,B 0,C 180,E1 -19787.013,E2 -19787.013} C_VEL
LIN {X 0,Y 234.744,Z 429.569,A -85,B 0,C 180,E1 -19788.341,E2 -19788.341} C_VEL
LIN {X 0,Y 235.235,Z 435.106,A -85,B 0,C 180,E1 -19789.02,E2 -19789.02} C_VEL
LIN {X 0,Y 234.682,Z 446.565,A -85,B 0,C 180,E1 -19790.737,E2 -19790.737} C_VEL
LIN {X 0,Y 234.193,Z 455.876,A -85,B 0,C 180,E1 -19792.499,E2 -19792.499} C_VEL
LIN {X 0,Y 233.984,Z 464.057,A -85,B 0,C 180,E1 -19794.398,E2 -19794.398} C_VEL
LIN {X 0,Y 233.507,Z 471.554,A -85,B 0,C 180,E1 -19796.549,E2 -19796.549} C_VEL
LIN {X 0,Y 233.372,Z 477.594,A -85,B 0,C 180,E1 -19798.706,E2 -19798.706} C_VEL
LIN {X 0,Y 233.568,Z 482.387,A -85,B 0,C 180,E1 -19800.862,E2 -19800.862} C_VEL
LIN {X 0,Y 234.124,Z 486.752,A -85,B 0,C 180,E1 -19803.442,E2 -19803.442} C_VEL
LIN {X 0,Y 234.784,Z 488.901,A -85,B 0,C 180,E1 -19805.152,E2 -19805.152} C_VEL
LIN {X 0,Y 235.681,Z 490.458,A -85,B 0,C 180,E1 -19806.851,E2 -19806.851} C_VEL
LIN {X 0,Y 236.805,Z 491.426,A -85,B 0,C 180,E1 -19808.534,E2 -19808.534} C_VEL
LIN {X 0,Y 238.146,Z 491.839,A -85,B 0,C 180,E1 -19810.199,E2 -19810.199} C_VEL
LIN {X 0,Y 239.859,Z 491.692,A -85,B 0,C 180,E1 -19811.836,E2 -19811.836} C_VEL
LIN {X 0,Y 241.647,Z 491.013,A -85,B 0,C 180,E1 -19813.454,E2 -19813.454} C_VEL
LIN {X 0,Y 243.683,Z 489.784,A -85,B 0,C 180,E1 -19815.044,E2 -19815.044} C_VEL
LIN {X 0,Y 247.045,Z 486.926,A -85,B 0,C 180,E1 -19817.38,E2 -19817.38} C_VEL
LIN {X 0,Y 250.883,Z 482.781,A -85,B 0,C 180,E1 -19819.643,E2 -19819.643} C_VEL
LIN {X 0,Y 255.116,Z 477.201,A -85,B 0,C 180,E1 -19821.833,E2 -19821.833} C_VEL
LIN {X 0,Y 256.467,Z 475.062,A -85,B 0,C 180,E1 -19822.56,E2 -19822.56} C_VEL
LIN {X 0,Y 257.837,Z 469.526,A -85,B 0,C 180,E1 -19824.988,E2 -19824.988} C_VEL
LIN {X 0,Y 258.499,Z 462.775,A -85,B 0,C 180,E1 -19828.007,E2 -19828.007} C_VEL
LIN {X 0,Y 258.514,Z 458.049,A -85,B 0,C 180,E1 -19830.341,E2 -19830.341} C_VEL
LIN {X 0,Y 258.318,Z 454.263,A -85,B 0,C 180,E1 -19832.497,E2 -19832.497} C_VEL
LIN {X 0,Y 257.739,Z 451.173,A -85,B 0,C 180,E1 -19834.934,E2 -19834.934} C_VEL
LIN {X 0,Y 257.103,Z 449.207,A -85,B 0,C 180,E1 -19837.559,E2 -19837.559} C_VEL
LIN {X 0,Y 256.926,Z 448.152,A -85,B 0,C 180,E1 -19840.011,E2 -19840.011} C_VEL
LIN {X 0,Y 257.115,Z 448.13,A -85,B 0,C 180,E1 -19842.436,E2 -19842.436} C_VEL
LIN {X 0,Y 257.624,Z 449.617,A -85,B 0,C 180,E1 -19845.177,E2 -19845.177} C_VEL
LIN {X 0,Y 259.06,Z 453.799,A -85,B 0,C 180,E1 -19848.87,E2 -19848.87} C_VEL
LIN {X 0,Y 260.123,Z 455.752,A -85,B 0,C 180,E1 -19850.328,E2 -19850.328} C_VEL
LIN {X 0,Y 261.815,Z 460.731,A -85,B 0,C 180,E1 -19852.879,E2 -19852.879} C_VEL
LIN {X 0,Y 262.088,Z 462.531,A -85,B 0,C 180,E1 -19853.558,E2 -19853.558} C_VEL
LIN {X 0,Y 261.637,Z 466.966,A -85,B 0,C 180,E1 -19854.683,E2 -19854.683} C_VEL
LIN {X 0,Y 260.671,Z 471.136,A -85,B 0,C 180,E1 -19855.585,E2 -19855.585} C_VEL
LIN {X 0,Y 258.833,Z 475.656,A -85,B 0,C 180,E1 -19856.35,E2 -19856.35} C_VEL
LIN {X 0,Y 254.045,Z 484.619,A -85,B 0,C 180,E1 -19857.789,E2 -19857.789} C_VEL
LIN {X 0,Y 251.149,Z 490.058,A -85,B 0,C 180,E1 -19858.941,E2 -19858.941} C_VEL
LIN {X 0,Y 246.773,Z 498.172,A -85,B 0,C 180,E1 -19861.043,E2 -19861.043} C_VEL
LIN {X 0,Y 242.02,Z 505.498,A -85,B 0,C 180,E1 -19863.249,E2 -19863.249} C_VEL
LIN {X 0,Y 237.992,Z 511.465,A -85,B 0,C 180,E1 -19865.579,E2 -19865.579} C_VEL
LIN {X 0,Y 234.442,Z 516.417,A -85,B 0,C 180,E1 -19867.993,E2 -19867.993} C_VEL
LIN {X 0,Y 230.781,Z 521.501,A -85,B 0,C 180,E1 -19871.351,E2 -19871.351} C_VEL
LIN {X 0,Y 228.775,Z 524.288,A -85,B 0,C 180,E1 -19873.949,E2 -19873.949} C_VEL
LIN {X 0,Y 226.915,Z 526.698,A -85,B 0,C 180,E1 -19877.478,E2 -19877.478} C_VEL
LIN {X 0,Y 226.297,Z 527.712,A -85,B 0,C 180,E1 -19881.066,E2 -19881.066} C_VEL
LIN {X 0,Y 226.383,Z 527.552,A -85,B 0,C 180,E1 -19883.431,E2 -19883.431} C_VEL
LIN {X 0,Y 226.79,Z 526.376,A -85,B 0,C 180,E1 -19886.446,E2 -19886.446} C_VEL
LIN {X 0,Y 227.237,Z 525.147,A -85,B 0,C 180,E1 -19888.227,E2 -19888.227} C_VEL
LIN {X 0,Y 227.562,Z 522.292,A -85,B 0,C 180,E1 -19890.884,E2 -19890.884} C_VEL
LIN {X 0,Y 227.637,Z 518.166,A -85,B 0,C 180,E1 -19893.54,E2 -19893.54} C_VEL
LIN {X 0,Y 227.61,Z 512.599,A -85,B 0,C 180,E1 -19896.204,E2 -19896.204} C_VEL
LIN {X 0,Y 227.53,Z 505.304,A -85,B 0,C 180,E1 -19898.884,E2 -19898.884} C_VEL
LIN {X 0,Y 227.795,Z 497.719,A -85,B 0,C 180,E1 -19901.117,E2 -19901.117} C_VEL
LIN {X 0,Y 228.254,Z 488.353,A -85,B 0,C 180,E1 -19903.351,E2 -19903.351} C_VEL
LIN {X 0,Y 229.027,Z 477.823,A -85,B 0,C 180,E1 -19905.347,E2 -19905.347} C_VEL
LIN {X 0,Y 229.268,Z 470.529,A -85,B 0,C 180,E1 -19906.471,E2 -19906.471} C_VEL
LIN {X 0,Y 228.369,Z 458.785,A -85,B 0,C 180,E1 -19907.923,E2 -19907.923} C_VEL
LIN {X 0,Y 227.673,Z 445.532,A -85,B 0,C 180,E1 -19909.146,E2 -19909.146} C_VEL
LIN {X 0,Y 227.732,Z 436.436,A -85,B 0,C 180,E1 -19909.786,E2 -19909.786} C_VEL
LIN {X 0,Y 229.949,Z 424.015,A -85,B 0,C 180,E1 -19916.306,E2 -19916.306} C_VEL
LIN {X 0,Y 232.272,Z 415.032,A -85,B 0,C 180,E1 -19920.956,E2 -19920.956} C_VEL
LIN {X 0,Y 232.295,Z 412.875,A -85,B 0,C 180,E1 -19922.099,E2 -19922.099} C_VEL
LIN {X 0,Y 230.554,Z 405.094,A -85,B 0,C 180,E1 -19926.376,E2 -19926.376} C_VEL
LIN {X 0,Y 228.778,Z 396.64,A -85,B 0,C 180,E1 -19931.243,E2 -19931.243} C_VEL
LIN {X 0,Y 227.939,Z 392.094,A -85,B 0,C 180,E1 -19933.97,E2 -19933.97} C_VEL
LIN {X 0,Y 227.819,Z 392.103,A -85,B 0,C 180,E1 -19937.763,E2 -19937.763} C_VEL
LIN {X 0,Y 227.87,Z 392.101,A -85,B 0,C 180,E1 -19941.914,E2 -19941.914} C_VEL
LIN {X 0,Y 227.891,Z 392.096,A -85,B 0,C 180,E1 -19946.373,E2 -19946.373} C_VEL
LIN {X 0,Y 227.905,Z 392.095,A -85,B 0,C 180,E1 -19950.436,E2 -19950.436} C_VEL
LIN {X 0,Y 227.929,Z 392.09,A -85,B 0,C 180,E1 -19954.426,E2 -19954.426} C_VEL
LIN {X 0,Y 227.963,Z 392.088,A -85,B 0,C 180,E1 -19958.287,E2 -19958.287} C_VEL
LIN {X 0,Y 228.035,Z 392.075,A -85,B 0,C 180,E1 -19962.826,E2 -19962.826} C_VEL
LIN {X 0,Y 228.095,Z 392.073,A -85,B 0,C 180,E1 -19967.544,E2 -19967.544} C_VEL
LIN {X 0,Y 228.326,Z 392.04,A -85,B 0,C 180,E1 -19971.147,E2 -19971.147} C_VEL
LIN {X 0,Y 228.359,Z 392.036,A -85,B 0,C 180,E1 -19972.929,E2 -19972.929} C_VEL
LIN {X 0,Y 228.558,Z 392.012,A -85,B 0,C 180,E1 -19978.238,E2 -19978.238} C_VEL
LIN {X 0,Y 228.556,Z 392.015,A -85,B 0,C 180,E1 -19981.762,E2 -19981.762} C_VEL
LIN {X 0,Y 228.359,Z 392.039,A -85,B 0,C 180,E1 -19987.071,E2 -19987.071} C_VEL
LIN {X 0,Y 228.172,Z 392.06,A -85,B 0,C 180,E1 -19990.65,E2 -19990.65} C_VEL
LIN {X 0,Y 228.059,Z 392.073,A -85,B 0,C 180,E1 -19996.102,E2 -19996.102} C_VEL
LIN {X 0,Y 227.943,Z 392.09,A -85,B 0,C 180,E1 -19999.825,E2 -19999.825} C_VEL
LIN {X 0,Y 227.915,Z 392.092,A -85,B 0,C 180,E1 -20003.633,E2 -20003.633} C_VEL
LIN {X 0,Y 227.887,Z 392.097,A -85,B 0,C 180,E1 -20007.555,E2 -20007.555} C_VEL
LIN {X 0,Y 227.871,Z 392.098,A -85,B 0,C 180,E1 -20011.622,E2 -20011.622} C_VEL
LIN {X 0,Y 227.881,Z 392.096,A -85,B 0,C 180,E1 -20015.872,E2 -20015.872} C_VEL
LIN {X 0,Y 227.827,Z 392.105,A -85,B 0,C 180,E1 -20020.377,E2 -20020.377} C_VEL
LIN {X 0,Y 227.836,Z 392.104,A -85,B 0,C 180,E1 -20025.192,E2 -20025.192} C_VEL
LIN {X 0,Y 227.835,Z 392.102,A -85,B 0,C 180,E1 -20029.625,E2 -20029.625} C_VEL
LIN {X 0,Y 227.901,Z 392.095,A -85,B 0,C 180,E1 -20034.132,E2 -20034.132} C_VEL
LIN {X 0,Y 227.874,Z 392.1,A -85,B 0,C 180,E1 -20038.379,E2 -20038.379} C_VEL
LIN {X 0,Y 227.886,Z 392.099,A -85,B 0,C 180,E1 -20042.445,E2 -20042.445} C_VEL
LIN {X 0,Y 227.926,Z 392.094,A -85,B 0,C 180,E1 -20046.369,E2 -20046.369} C_VEL
LIN {X 0,Y 227.957,Z 392.088,A -85,B 0,C 180,E1 -20050.176,E2 -20050.176} C_VEL
LIN {X 0,Y 228.06,Z 392.077,A -85,B 0,C 180,E1 -20053.898,E2 -20053.898} C_VEL
LIN {X 0,Y 228.097,Z 392.067,A -85,B 0,C 180,E1 -20057.545,E2 -20057.545} C_VEL
LIN {X 0,Y 228.307,Z 392.044,A -85,B 0,C 180,E1 -20061.146,E2 -20061.146} C_VEL
LIN {X 0,Y 228.356,Z 392.038,A -85,B 0,C 180,E1 -20062.929,E2 -20062.929} C_VEL
LIN {X 0,Y 228.557,Z 392.015,A -85,B 0,C 180,E1 -20068.238,E2 -20068.238} C_VEL
LIN {X 0,Y 228.557,Z 392.015,A -85,B 0,C 180,E1 -20071.762,E2 -20071.762} C_VEL
LIN {X 0,Y 228.327,Z 392.041,A -85,B 0,C 180,E1 -20077.073,E2 -20077.073} C_VEL
LIN {X 0,Y 228.148,Z 392.063,A -85,B 0,C 180,E1 -20080.651,E2 -20080.651} C_VEL
LIN {X 0,Y 228.068,Z 392.074,A -85,B 0,C 180,E1 -20084.272,E2 -20084.272} C_VEL
LIN {X 0,Y 228.006,Z 392.083,A -85,B 0,C 180,E1 -20087.953,E2 -20087.953} C_VEL
LIN {X 0,Y 227.933,Z 392.089,A -85,B 0,C 180,E1 -20092.33,E2 -20092.33} C_VEL
LIN {X 0,Y 227.945,Z 392.089,A -85,B 0,C 180,E1 -20096.603,E2 -20096.603} C_VEL
LIN {X 0,Y 227.911,Z 392.091,A -85,B 0,C 180,E1 -20100.296,E2 -20100.296} C_VEL
LIN {X 0,Y 227.893,Z 392.098,A -85,B 0,C 180,E1 -20103.718,E2 -20103.718} C_VEL
LIN {X 0,Y 227.872,Z 392.095,A -85,B 0,C 180,E1 -20108.086,E2 -20108.086} C_VEL
LIN {X 0,Y 227.818,Z 392.106,A -85,B 0,C 180,E1 -20112.741,E2 -20112.741} C_VEL
LIN {X 0,Y 227.815,Z 392.106,A -85,B 0,C 180,E1 -20117.258,E2 -20117.258} C_VEL
LIN {X 0,Y 227.854,Z 392.101,A -85,B 0,C 180,E1 -20121.911,E2 -20121.911} C_VEL
LIN {X 0,Y 228.024,Z 392.075,A -85,B 0,C 180,E1 -20126.324,E2 -20126.324} C_VEL
LIN {X 0,Y 228.187,Z 392.153,A -85,B 0,C 180,E1 -20127.907,E2 -20127.907} C_VEL
LIN {X 0,Y 228.288,Z 394.131,A -85,B 0,C 180,E1 -20129.543,E2 -20129.543} C_VEL
LIN {X 0,Y 227.751,Z 399.032,A -85,B 0,C 180,E1 -20133.495,E2 -20133.495} C_VEL
LIN {X 0,Y 227.184,Z 405.017,A -85,B 0,C 180,E1 -20138.209,E2 -20138.209} C_VEL
LIN {X 0,Y 226.755,Z 411.084,A -85,B 0,C 180,E1 -20142.876,E2 -20142.876} C_VEL
LIN {X 0,Y 226.504,Z 416.591,A -85,B 0,C 180,E1 -20147.057,E2 -20147.057} C_VEL
LIN {X 0,Y 227.642,Z 429.8,A -85,B 0,C 180,E1 -20148.424,E2 -20148.424} C_VEL
LIN {X 0,Y 228.128,Z 435.337,A -85,B 0,C 180,E1 -20149.123,E2 -20149.123} C_VEL
LIN {X 0,Y 227.594,Z 446.869,A -85,B 0,C 180,E1 -20150.894,E2 -20150.894} C_VEL
LIN {X 0,Y 227.067,Z 457.057,A -85,B 0,C 180,E1 -20152.888,E2 -20152.888} C_VEL
LIN {X 0,Y 226.839,Z 464.479,A -85,B 0,C 180,E1 -20154.667,E2 -20154.667} C_VEL
LIN {X 0,Y 226.388,Z 471.955,A -85,B 0,C 180,E1 -20156.886,E2 -20156.886} C_VEL
LIN {X 0,Y 226.319,Z 479.095,A -85,B 0,C 180,E1 -20159.555,E2 -20159.555} C_VEL
LIN {X 0,Y 226.6,Z 483.776,A -85,B 0,C 180,E1 -20161.777,E2 -20161.777} C_VEL
LIN {X 0,Y 227.363,Z 487.976,A -85,B 0,C 180,E1 -20164.432,E2 -20164.432} C_VEL
LIN {X 0,Y 228.668,Z 490.826,A -85,B 0,C 180,E1 -20167.062,E2 -20167.062} C_VEL
LIN {X 0,Y 229.825,Z 492.044,A -85,B 0,C 180,E1 -20168.795,E2 -20168.795} C_VEL
LIN {X 0,Y 231.21,Z 492.679,A -85,B 0,C 180,E1 -20170.508,E2 -20170.508} C_VEL
LIN {X 0,Y 232.982,Z 492.749,A -85,B 0,C 180,E1 -20172.19,E2 -20172.19} C_VEL
LIN {X 0,Y 234.858,Z 492.319,A -85,B 0,C 180,E1 -20173.851,E2 -20173.851} C_VEL
LIN {X 0,Y 236.975,Z 491.319,A -85,B 0,C 180,E1 -20175.481,E2 -20175.481} C_VEL
LIN {X 0,Y 240.494,Z 488.864,A -85,B 0,C 180,E1 -20177.869,E2 -20177.869} C_VEL
LIN {X 0,Y 244.495,Z 485.147,A -85,B 0,C 180,E1 -20180.178,E2 -20180.178} C_VEL
LIN {X 0,Y 248.902,Z 480.095,A -85,B 0,C 180,E1 -20182.407,E2 -20182.407} C_VEL
LIN {X 0,Y 250.464,Z 478.098,A -85,B 0,C 180,E1 -20183.131,E2 -20183.131} C_VEL
LIN {X 0,Y 251.76,Z 474.643,A -85,B 0,C 180,E1 -20184.755,E2 -20184.755} C_VEL
LIN {X 0,Y 253.05,Z 468.706,A -85,B 0,C 180,E1 -20187.674,E2 -20187.674} C_VEL
LIN {X 0,Y 253.577,Z 464.387,A -85,B 0,C 180,E1 -20189.926,E2 -20189.926} C_VEL
LIN {X 0,Y 253.822,Z 459.943,A -85,B 0,C 180,E1 -20192.566,E2 -20192.566} C_VEL
LIN {X 0,Y 253.729,Z 458.298,A -85,B 0,C 180,E1 -20193.801,E2 -20193.801} C_VEL
LIN {X 0,Y 253.351,Z 455.881,A -85,B 0,C 180,E1 -20196.441,E2 -20196.441} C_VEL
LIN {X 0,Y 253.23,Z 454.333,A -85,B 0,C 180,E1 -20199.667,E2 -20199.667} C_VEL
LIN {X 0,Y 253.395,Z 454.128,A -85,B 0,C 180,E1 -20201.732,E2 -20201.732} C_VEL
LIN {X 0,Y 253.67,Z 454.932,A -85,B 0,C 180,E1 -20203.917,E2 -20203.917} C_VEL
LIN {X 0,Y 254.201,Z 456.847,A -85,B 0,C 180,E1 -20206.275,E2 -20206.275} C_VEL
LIN {X 0,Y 256.074,Z 461.71,A -85,B 0,C 180,E1 -20210.216,E2 -20210.216} C_VEL
LIN {X 0,Y 257.242,Z 465.754,A -85,B 0,C 180,E1 -20212.401,E2 -20212.401} C_VEL
LIN {X 0,Y 257.259,Z 467.55,A -85,B 0,C 180,E1 -20213.057,E2 -20213.057} C_VEL
LIN {X 0,Y 255.645,Z 475.824,A -85,B 0,C 180,E1 -20215.267,E2 -20215.267} C_VEL
LIN {X 0,Y 253.27,Z 484.492,A -85,B 0,C 180,E1 -20217.518,E2 -20217.518} C_VEL
LIN {X 0,Y 251.149,Z 490.058,A -85,B 0,C 180,E1 -20218.941,E2 -20218.941} C_VEL
LIN {X 0,Y 248.697,Z 493.992,A -85,B 0,C 180,E1 -20219.809,E2 -20219.809} C_VEL
LIN {X 0,Y 245.305,Z 497.816,A -85,B 0,C 180,E1 -20220.535,E2 -20220.535} C_VEL
LIN {X 0,Y 236.714,Z 505.849,A -85,B 0,C 180,E1 -20222.303,E2 -20222.303} C_VEL
LIN {X 0,Y 234.051,Z 508.808,A -85,B 0,C 180,E1 -20223.353,E2 -20223.353} C_VEL
LIN {X 0,Y 230.308,Z 513.802,A -85,B 0,C 180,E1 -20225.672,E2 -20225.672} C_VEL
LIN {X 0,Y 226.806,Z 518.048,A -85,B 0,C 180,E1 -20228.17,E2 -20228.17} C_VEL
LIN {X 0,Y 224.872,Z 520.412,A -85,B 0,C 180,E1 -20229.892,E2 -20229.892} C_VEL
LIN {X 0,Y 221.917,Z 523.934,A -85,B 0,C 180,E1 -20233.439,E2 -20233.439} C_VEL
LIN {X 0,Y 219.956,Z 526.051,A -85,B 0,C 180,E1 -20237.075,E2 -20237.075} C_VEL
LIN {X 0,Y 219.296,Z 526.723,A -85,B 0,C 180,E1 -20240.779,E2 -20240.779} C_VEL
LIN {X 0,Y 219.489,Z 525.986,A -85,B 0,C 180,E1 -20244.487,E2 -20244.487} C_VEL
LIN {X 0,Y 219.806,Z 525.002,A -85,B 0,C 180,E1 -20246.333,E2 -20246.333} C_VEL
LIN {X 0,Y 220.291,Z 523.616,A -85,B 0,C 180,E1 -20248.171,E2 -20248.171} C_VEL
LIN {X 0,Y 220.606,Z 521.738,A -85,B 0,C 180,E1 -20250,E2 -20250} C_VEL
LIN {X 0,Y 220.734,Z 517.807,A -85,B 0,C 180,E1 -20252.737,E2 -20252.737} C_VEL
LIN {X 0,Y 220.67,Z 512.406,A -85,B 0,C 180,E1 -20255.482,E2 -20255.482} C_VEL
LIN {X 0,Y 220.563,Z 505.202,A -85,B 0,C 180,E1 -20258.299,E2 -20258.299} C_VEL
LIN {X 0,Y 220.803,Z 498.01,A -85,B 0,C 180,E1 -20260.545,E2 -20260.545} C_VEL
LIN {X 0,Y 221.19,Z 488.893,A -85,B 0,C 180,E1 -20262.851,E2 -20262.851} C_VEL
LIN {X 0,Y 221.893,Z 478.702,A -85,B 0,C 180,E1 -20264.912,E2 -20264.912} C_VEL
LIN {X 0,Y 222.319,Z 471.893,A -85,B 0,C 180,E1 -20266.058,E2 -20266.058} C_VEL
LIN {X 0,Y 221.34,Z 459.254,A -85,B 0,C 180,E1 -20267.718,E2 -20267.718} C_VEL
LIN {X 0,Y 220.669,Z 447.006,A -85,B 0,C 180,E1 -20268.932,E2 -20268.932} C_VEL
LIN {X 0,Y 220.624,Z 436.12,A -85,B 0,C 180,E1 -20269.783,E2 -20269.783} C_VEL
LIN {X 0,Y 222.761,Z 424.347,A -85,B 0,C 180,E1 -20276.212,E2 -20276.212} C_VEL
LIN {X 0,Y 225.13,Z 415.453,A -85,B 0,C 180,E1 -20281.003,E2 -20281.003} C_VEL
LIN {X 0,Y 225.041,Z 412.709,A -85,B 0,C 180,E1 -20282.52,E2 -20282.52} C_VEL
LIN {X 0,Y 223.162,Z 404.296,A -85,B 0,C 180,E1 -20287.34,E2 -20287.34} C_VEL
LIN {X 0,Y 221.425,Z 395.826,A -85,B 0,C 180,E1 -20292.411,E2 -20292.411} C_VEL
LIN {X 0,Y 220.903,Z 392.968,A -85,B 0,C 180,E1 -20294.192,E2 -20294.192} C_VEL
LIN {X 0,Y 220.801,Z 392.98,A -85,B 0,C 180,E1 -20299.81,E2 -20299.81} C_VEL
LIN {X 0,Y 220.832,Z 392.975,A -85,B 0,C 180,E1 -20302.794,E2 -20302.794} C_VEL
LIN {X 0,Y 220.824,Z 392.975,A -85,B 0,C 180,E1 -20307.245,E2 -20307.245} C_VEL
LIN {X 0,Y 220.828,Z 392.977,A -85,B 0,C 180,E1 -20311.485,E2 -20311.485} C_VEL
LIN {X 0,Y 220.868,Z 392.97,A -85,B 0,C 180,E1 -20315.565,E2 -20315.565} C_VEL
LIN {X 0,Y 220.893,Z 392.97,A -85,B 0,C 180,E1 -20319.514,E2 -20319.514} C_VEL
LIN {X 0,Y 221.017,Z 392.95,A -85,B 0,C 180,E1 -20323.37,E2 -20323.37} C_VEL
LIN {X 0,Y 221.118,Z 392.94,A -85,B 0,C 180,E1 -20329.006,E2 -20329.006} C_VEL
LIN {X 0,Y 221.312,Z 392.914,A -85,B 0,C 180,E1 -20332.702,E2 -20332.702} C_VEL
LIN {X 0,Y 221.516,Z 392.889,A -85,B 0,C 180,E1 -20338.182,E2 -20338.182} C_VEL
LIN {X 0,Y 221.514,Z 392.891,A -85,B 0,C 180,E1 -20341.818,E2 -20341.818} C_VEL
LIN {X 0,Y 221.312,Z 392.917,A -85,B 0,C 180,E1 -20347.298,E2 -20347.298} C_VEL
LIN {X 0,Y 221.118,Z 392.94,A -85,B 0,C 180,E1 -20350.994,E2 -20350.994} C_VEL
LIN {X 0,Y 221.017,Z 392.951,A -85,B 0,C 180,E1 -20356.63,E2 -20356.63} C_VEL
LIN {X 0,Y 220.893,Z 392.968,A -85,B 0,C 180,E1 -20360.486,E2 -20360.486} C_VEL
LIN {X 0,Y 220.868,Z 392.97,A -85,B 0,C 180,E1 -20364.435,E2 -20364.435} C_VEL
LIN {X 0,Y 220.837,Z 392.975,A -85,B 0,C 180,E1 -20368.514,E2 -20368.514} C_VEL
LIN {X 0,Y 220.818,Z 392.979,A -85,B 0,C 180,E1 -20372.756,E2 -20372.756} C_VEL
LIN {X 0,Y 220.811,Z 392.979,A -85,B 0,C 180,E1 -20377.279,E2 -20377.279} C_VEL
LIN {X 0,Y 220.771,Z 392.981,A -85,B 0,C 180,E1 -20381.952,E2 -20381.952} C_VEL
LIN {X 0,Y 220.777,Z 392.982,A -85,B 0,C 180,E1 -20385.547,E2 -20385.547} C_VEL
LIN {X 0,Y 220.81,Z 392.979,A -85,B 0,C 180,E1 -20390.464,E2 -20390.464} C_VEL
LIN {X 0,Y 220.833,Z 392.977,A -85,B 0,C 180,E1 -20392.795,E2 -20392.795} C_VEL
LIN {X 0,Y 220.826,Z 392.976,A -85,B 0,C 180,E1 -20397.246,E2 -20397.246} C_VEL
